// TIA Portal V20 export
FUNCTION_BLOCK "CallEquipment"   // FB21, LAD
TITLE = CallEquipment
AUTHOR : ERsystem_FA2_DH. Kim
// This block contains the logic and futher calls (e.g. sequences, control modules, diagnostics etc.) of the equipment module.
// stored: IsIECCheckEnabled true, MemoryReserve 100, Namespace Unit1.Em6, SetENOAutomatically false
   VAR_INPUT
      ZoneOperationEnable { ExternalWritable := 'False'} : "LWONIK_typeSafetyZoneManualOperation";
   END_VAR
   VAR_IN_OUT
      unitStatus : "LAF_typeUnitStatus";   // Current unit status o be used in this EM
      unitAlarmDB : "LAF_typeAlarms";   // Summarized EM Alarms for the Unit
      emFeedback : "LUC_typeEmFeedback";   // Feedback of the EM to the Unit
   END_VAR
   VAR
      InstSequenceStackTable { S7_SetPoint := 'True'} : "Unit1.Em6.Sequence_1_StackTable";
      InstSequenceGaugeRnR { S7_SetPoint := 'True'} : "Unit1.Em6.Sequence_10_GaugeRnR";
      InstSequenceUtility { S7_SetPoint := 'True'} : "Unit1.Em6.Sequence_20_Utility";
      instStackTableHomeJob1 { S7_SetPoint := 'True'} : "LAF_SelectJob";
      instStackTableMotionAutoJob2 { S7_SetPoint := 'True'} : "LAF_SelectJob";
      instStackTableRollerMoveJob12 { S7_SetPoint := 'True'} : "LAF_SelectJob";
      instStackTableRollerMoveJob13 { S7_SetPoint := 'True'} : "LAF_SelectJob";
      instStackTableAnodeMendrelJob22 { S7_SetPoint := 'True'} : "LAF_SelectJob";
      instStackTableCathodeMendrelJob23 { S7_SetPoint := 'True'} : "LAF_SelectJob";
      instStackTableVisionJob30 { S7_SetPoint := 'True'} : "LAF_SelectJob";
      instStackTableDownJob31 { S7_SetPoint := 'True'} : "LAF_SelectJob";
      instStackTableUnloadJob4 { S7_SetPoint := 'True'} : "LAF_SelectJob";
      instGaugeRnRReadyJob1 { S7_SetPoint := 'True'} : "LAF_SelectJob";
      instGaugeRnRVaccumJob2 { S7_SetPoint := 'True'} : "LAF_SelectJob";
      instGaugeRnRVisionJob3 { S7_SetPoint := 'True'} : "LAF_SelectJob";
      instGaugeRnRBlowJob4 { S7_SetPoint := 'True'} : "LAF_SelectJob";
      instUtilityFinalRollerHomeJob1 { S7_SetPoint := 'True'} : "LAF_SelectJob";
      instUtilityStackTableOutHomeJob2 { S7_SetPoint := 'True'} : "LAF_SelectJob";
      instUtilityAllMendrelOpenJob3 { S7_SetPoint := 'True'} : "LAF_SelectJob";
      instUtilityAllMendrelCloseJob4 { S7_SetPoint := 'True'} : "LAF_SelectJob";
      instCmStackTableElectrodeDetectSensor { S7_SetPoint := 'True'} : "LBC_DigitalSignalCn";
      instCmMasterVirtualAxisX : "LBC_Axis64Pos_TecPlcCn";
      instCmFinalRollerFrontAxisX : "LBC_Axis64Pos_TecPlcCn";
      instCmFinalRollerRearAxisX { S7_SetPoint := 'True'} : "LBC_Axis64Pos_TecPlcCn";
      instCmMendrelAnodeFrontAxisY { S7_SetPoint := 'True'} : "LBC_Axis64Pos_TecPlcCn";
      instCmMendrelAnodeFrontAxisZ { S7_SetPoint := 'True'} : "LBC_Axis64Pos_TecPlcCn";
      instCmMendrelAnodeRearAxisY { S7_SetPoint := 'True'} : "LBC_Axis64Pos_TecPlcCn";
      instCmMendrelAnodeRearAxisZ { S7_SetPoint := 'True'} : "LBC_Axis64Pos_TecPlcCn";
      instCmMendrelCathodeFrontAxisY { S7_SetPoint := 'True'} : "LBC_Axis64Pos_TecPlcCn";
      instCmMendrelCathodeFrontAxisZ { S7_SetPoint := 'True'} : "LBC_Axis64Pos_TecPlcCn";
      instCmMendrelCathodeRearAxisY { S7_SetPoint := 'True'} : "LBC_Axis64Pos_TecPlcCn";
      instCmMendrelCathodeRearAxisZ { S7_SetPoint := 'True'} : "LBC_Axis64Pos_TecPlcCn";
      instCmStackTableAxisZ { ExternalAccessible := 'False'; ExternalVisible := 'False'; ExternalWritable := 'False'; S7_SetPoint := 'True'} : "LBC_Axis64Pos_TecPlcCn";
      instCmStackTableOutFrontAxisZ { ExternalAccessible := 'False'; ExternalVisible := 'False'; ExternalWritable := 'False'; S7_SetPoint := 'True'} : "LBC_Axis64Pos_TecPlcCn";
      instCmStackTableOutRearAxisZ { ExternalAccessible := 'False'; ExternalVisible := 'False'; ExternalWritable := 'False'; S7_SetPoint := 'True'} : "LBC_Axis64Pos_TecPlcCn";
      instInterlockFinalRollerFrontAxisX : "LER_Axis64Pos_InterlockSummary";
      instInterlockFinalRollerRearAxisX : "LER_Axis64Pos_InterlockSummary";
      instInterlockMendrelAnodeFrontAxisY : "LER_Axis64Pos_InterlockSummary";
      instInterlockMendrelAnodeFrontAxisZ : "LER_Axis64Pos_InterlockSummary";
      instInterlockMendrelAnodeRearAxisY : "LER_Axis64Pos_InterlockSummary";
      instInterlockMendrelAnodeRearAxisZ : "LER_Axis64Pos_InterlockSummary";
      instInterlockMendrelCathodeFrontAxisY : "LER_Axis64Pos_InterlockSummary";
      instInterlockMendrelCathodeFrontAxisZ : "LER_Axis64Pos_InterlockSummary";
      instInterlockMendrelCathodeRearAxisY : "LER_Axis64Pos_InterlockSummary";
      instInterlockMendrelCathodeRearAxisZ : "LER_Axis64Pos_InterlockSummary";
      instInterlockStackTableAxisZ : "LER_Axis64Pos_InterlockSummary";
      instInterlockStackTableOutFrontAxisZ : "LER_Axis64Pos_InterlockSummary";
      instInterlockStackTableOutRearAxisZ : "LER_Axis64Pos_InterlockSummary";
      instFinalRollerFrontAxisXMCGearIn { S7_SetPoint := 'True'} : MC_GEARIN;
      instFinalRollerRearAxisXMCGearIn { S7_SetPoint := 'True'} : MC_GEARIN;
      instStackTableOutFrontAxisZMCGearIn { S7_SetPoint := 'True'} : MC_GEARIN;
      instStackTableOutRearAxisZMCGearIn { S7_SetPoint := 'True'} : MC_GEARIN;
      instFinalRollerFrontAxisXMCWirteParameter { S7_SetPoint := 'True'} : MC_WRITEPARAMETER;
      instFinalRollerRearAxisXMCWirteParameter { S7_SetPoint := 'True'} : MC_WRITEPARAMETER;
      instStackTableOutFrontAxisZMCWirteParameter { S7_SetPoint := 'True'} : MC_WRITEPARAMETER;
      instStackTableOutRearAxisZMCWirteParameter { S7_SetPoint := 'True'} : MC_WRITEPARAMETER;
      instCmMendrelCathodeFrontClamp { ExternalAccessible := 'False'; ExternalVisible := 'False'; ExternalWritable := 'False'; S7_SetPoint := 'True'} : "LBC_TwoWayActuatorCn";
      instCmMendrelAnodeFrontClamp { ExternalAccessible := 'False'; ExternalVisible := 'False'; ExternalWritable := 'False'; S7_SetPoint := 'True'} : "LBC_TwoWayActuatorCn";
      instCmMendrelCathodeRearClamp { ExternalAccessible := 'False'; ExternalVisible := 'False'; ExternalWritable := 'False'; S7_SetPoint := 'True'} : "LBC_TwoWayActuatorCn";
      instCmMendrelAnodeRearClamp { ExternalAccessible := 'False'; ExternalVisible := 'False'; ExternalWritable := 'False'; S7_SetPoint := 'True'} : "LBC_TwoWayActuatorCn";
      instcmStackTableVaccum { ExternalAccessible := 'False'; ExternalVisible := 'False'; ExternalWritable := 'False'; S7_SetPoint := 'True'} : "LBC_TwoWayActuatorCn";
      instcmStackTableGapPadUpDown { ExternalAccessible := 'False'; ExternalVisible := 'False'; ExternalWritable := 'False'; S7_SetPoint := 'True'} : "LBC_TwoWayActuatorCn";
      instCmStackTableVisionControllerInterface : "LER_Vision_XGX2000";
      instGapVisionConversion : "LER_StackTableVisionConversion";
      instManageAlarms { ExternalWritable := 'False'} : "LAF_ManageAlarms";
      instEventsPFE : "Unit1.Em6.EventsPFE";
      instLER_BrakeTestMendrelAnodeFrontAxisZ : "LER_BrakeTest";
      instLER_BrakeTestMendrelAnodeRearAxisZ { S7_SetPoint := 'True'} : "LER_BrakeTest";
      instLER_BrakeTestMendrelCathodeFrontAxisZ { S7_SetPoint := 'True'} : "LER_BrakeTest";
      instLER_BrakeTestMendrelCathodeRearAxisZ { S7_SetPoint := 'True'} : "LER_BrakeTest";
      instLER_BrakeTestStackTableAxisZ { S7_SetPoint := 'True'} : "LER_BrakeTest";
      instLER_BrakeTestStackTableOutFrontAxisZ { S7_SetPoint := 'True'} : "LER_BrakeTest";
      instLER_BrakeTestStackTableOutRearAxisZ { S7_SetPoint := 'True'} : "LER_BrakeTest";
      statUnitStatus { ExternalWritable := 'False'} : "LAF_typeUnitStatus";   // Unit Status used in this EM
      statSlmStatus : Struct
         running { ExternalWritable := 'False'} : Bool;
         powerOff { ExternalWritable := 'False'} : Bool;
      END_STRUCT;
      statAllBrakeTest { ExternalWritable := 'False'} : "LER_typeBrakeTestUnitCommands";
      statTonTime { ExternalAccessible := 'False'; ExternalVisible := 'False'; ExternalWritable := 'False'} : Array[0..1999] of TON_TIME;
      statTofTime { ExternalAccessible := 'False'; ExternalVisible := 'False'; ExternalWritable := 'False'} : Array[0..99] of TOF_TIME;
      statLReal { ExternalAccessible := 'False'; ExternalVisible := 'False'; ExternalWritable := 'False'} : Array[0..99] of LReal;
      statPulse { ExternalAccessible := 'False'; ExternalVisible := 'False'; ExternalWritable := 'False'} : Struct
         miscellaneous : Array[0..99] of Bool;
         workingDone : Array[0..99] of Bool;
         axisEnable : Array[0..99] of Bool;
         brakeTest : Array[0..99] of Bool;
      END_STRUCT;
      statEnableManualCmds : Bool;
      scan_on : Bool;
      "*** Interlock Axis ***" { ExternalAccessible := 'False'; ExternalVisible := 'False'; ExternalWritable := 'False'} : Bool;
      instFinalRollerFrontAxisX_CW { S7_SetPoint := 'True'} : "Jog.LER_Axis";
      instFinalRollerFrontAxisX_CCW { S7_SetPoint := 'True'} : "Jog.LER_Axis";
      instFinalRollerFrontAxisX_Home { S7_SetPoint := 'True'} : "Homing.LER_Axis";
      instFinalRollerFrontAxisX_Position { S7_SetPoint := 'True'} : Array[0..6] of "Position.LER_Axis";
      instFinalRollerRearAxisX_CW { S7_SetPoint := 'True'} : "Jog.LER_Axis";
      instFinalRollerRearAxisX_CCW { S7_SetPoint := 'True'} : "Jog.LER_Axis";
      instFinalRollerRearAxisX_Home { S7_SetPoint := 'True'} : "Homing.LER_Axis";
      instFinalRollerRearAxisX_Position { S7_SetPoint := 'True'} : Array[0..6] of "Position.LER_Axis";
      instMendrelAnodeFrontAxisY_CW { S7_SetPoint := 'True'} : "Jog.LER_Axis";
      instMendrelAnodeFrontAxisY_CCW { S7_SetPoint := 'True'} : "Jog.LER_Axis";
      instMendrelAnodeFrontAxisY_Home { S7_SetPoint := 'True'} : "Homing.LER_Axis";
      instMendrelAnodeFrontAxisY_Position { S7_SetPoint := 'True'} : Array[0..15] of "Position.LER_Axis";
      instMendrelAnodeFrontAxisZ_CW { S7_SetPoint := 'True'} : "Jog.LER_Axis";
      instMendrelAnodeFrontAxisZ_CCW { S7_SetPoint := 'True'} : "Jog.LER_Axis";
      instMendrelAnodeFrontAxisZ_Home { S7_SetPoint := 'True'} : "Homing.LER_Axis";
      instMendrelAnodeFrontAxisZ_Position { S7_SetPoint := 'True'} : Array[0..6] of "Position.LER_Axis";
      instMendrelAnodeRearAxisY_CW { S7_SetPoint := 'True'} : "Jog.LER_Axis";
      instMendrelAnodeRearAxisY_CCW { S7_SetPoint := 'True'} : "Jog.LER_Axis";
      instMendrelAnodeRearAxisY_Home { S7_SetPoint := 'True'} : "Homing.LER_Axis";
      instMendrelAnodeRearAxisY_Position { S7_SetPoint := 'True'} : Array[0..6] of "Position.LER_Axis";
      instMendrelAnodeRearAxisZ_CW { S7_SetPoint := 'True'} : "Jog.LER_Axis";
      instMendrelAnodeRearAxisZ_CCW { S7_SetPoint := 'True'} : "Jog.LER_Axis";
      instMendrelAnodeRearAxisZ_Home { S7_SetPoint := 'True'} : "Homing.LER_Axis";
      instMendrelAnodeRearAxisZ_Position { S7_SetPoint := 'True'} : Array[0..6] of "Position.LER_Axis";
      instMendrelCathodeFrontAxisY_CW { S7_SetPoint := 'True'} : "Jog.LER_Axis";
      instMendrelCathodeFrontAxisY_CCW { S7_SetPoint := 'True'} : "Jog.LER_Axis";
      instMendrelCathodeFrontAxisY_Home { S7_SetPoint := 'True'} : "Homing.LER_Axis";
      instMendrelCathodeFrontAxisY_Position { S7_SetPoint := 'True'} : Array[0..6] of "Position.LER_Axis";
      instMendrelCathodeFrontAxisZ_CW { S7_SetPoint := 'True'} : "Jog.LER_Axis";
      instMendrelCathodeFrontAxisZ_CCW { S7_SetPoint := 'True'} : "Jog.LER_Axis";
      instMendrelCathodeFrontAxisZ_Home { S7_SetPoint := 'True'} : "Homing.LER_Axis";
      instMendrelCathodeFrontAxisZ_Position { S7_SetPoint := 'True'} : Array[0..6] of "Position.LER_Axis";
      instMendrelCathodeRearAxisY_CW { S7_SetPoint := 'True'} : "Jog.LER_Axis";
      instMendrelCathodeRearAxisY_CCW { S7_SetPoint := 'True'} : "Jog.LER_Axis";
      instMendrelCathodeRearAxisY_Home { S7_SetPoint := 'True'} : "Homing.LER_Axis";
      instMendrelCathodeRearAxisY_Position { S7_SetPoint := 'True'} : Array[0..6] of "Position.LER_Axis";
      instMendrelCathodeRearAxisZ_CW { S7_SetPoint := 'True'} : "Jog.LER_Axis";
      instMendrelCathodeRearAxisZ_CCW { S7_SetPoint := 'True'} : "Jog.LER_Axis";
      instMendrelCathodeRearAxisZ_Home { S7_SetPoint := 'True'} : "Homing.LER_Axis";
      instMendrelCathodeRearAxisZ_Position { S7_SetPoint := 'True'} : Array[0..6] of "Position.LER_Axis";
      instStackTableAxisZ_CW { S7_SetPoint := 'True'} : "Jog.LER_Axis";
      instStackTableAxisZ_CCW { S7_SetPoint := 'True'} : "Jog.LER_Axis";
      instStackTableAxisZ_Home { S7_SetPoint := 'True'} : "Homing.LER_Axis";
      instStackTableAxisZ_Position { S7_SetPoint := 'True'} : Array[0..6] of "Position.LER_Axis";
      instStackTableOutFrontAxisZ_CW { S7_SetPoint := 'True'} : "Jog.LER_Axis";
      instStackTableOutFrontAxisZ_CCW { S7_SetPoint := 'True'} : "Jog.LER_Axis";
      instStackTableOutFrontAxisZ_Home { S7_SetPoint := 'True'} : "Homing.LER_Axis";
      instStackTableOutFrontAxisZ_Position { S7_SetPoint := 'True'} : Array[0..6] of "Position.LER_Axis";
      instStackTableOutRearAxisZ_CW { S7_SetPoint := 'True'} : "Jog.LER_Axis";
      instStackTableOutRearAxisZ_CCW { S7_SetPoint := 'True'} : "Jog.LER_Axis";
      instStackTableOutRearAxisZ_Home { S7_SetPoint := 'True'} : "Homing.LER_Axis";
      instStackTableOutRearAxisZ_Position { S7_SetPoint := 'True'} : Array[0..6] of "Position.LER_Axis";
      "*** Interlock Actuator ******" { ExternalAccessible := 'False'; ExternalVisible := 'False'; ExternalWritable := 'False'} : Bool;
      instCmMendrelCathodeFrontClampInterlock : Array[0..1] of "Cylinder.LER_Actuator";
      instCmMendrelAnodeFrontClampInterlock { S7_SetPoint := 'True'} : Array[0..1] of "Cylinder.LER_Actuator";
      instCmMendrelCathodeRearClampInterlock { S7_SetPoint := 'True'} : Array[0..1] of "Cylinder.LER_Actuator";
      instCmMendrelAnodeRearClampInterlock { S7_SetPoint := 'True'} : Array[0..1] of "Cylinder.LER_Actuator";
      instcmStackTableVaccumInterlock { S7_SetPoint := 'True'} : Array[0..1] of "Cylinder.LER_Actuator";
      instcmStackTableGapPadUpDownInterlock { S7_SetPoint := 'True'} : Array[0..1] of "Cylinder.LER_Actuator";
      AXIS21 : "LER_CM_Name";
      AXIS26 : "LER_CM_Name";
      AXIS31 : "LER_CM_Name";
      Cylinder33 : "LER_CM_Name";
      Vaccum20 : "LER_CM_Name";
      instFinalRollerGearInVel : MC_GEARINVELOCITY;
      instStackTableOutGearInVel : MC_GEARINVELOCITY;
      instFinalRollerGantryHoming : "LER_GantryHoming";
      instStackTableOutGantryHoming : "LER_GantryHoming";
      citi_Ptrig : Array[0..20] of Bool;
      citiTon : Array[0..20] of TON_TIME;
      citi : Time;
      citiTest : Array[0..20] of Bool;
   END_VAR
   VAR_TEMP
      tempIndex : Int;
      tempScInProduction : Bool;   // Mode Production and StateComplete
      tempScNoProduction : Bool;   // Mode Manual and StateComplete
   END_VAR
   VAR CONSTANT
      delayTime : Time := T#3s;
      TRUE : Bool := TRUE;
      FALSE : Bool := FALSE;
      NO_JOB : DInt;   // No job
      MIN_POSITION_NUMBER : SInt;
      INIT_POSITION_NUMBER : SInt := -1;
   END_VAR
   // // statPulse.brakeTest[0] : Unit Mode Production Rising Edge
   // // statPulse.brakeTest[1] : Unit Mode Production Rising Edge Old
   // // statPulse.brakeTest[10] : Mendrel Anode Front Z Axis Error Pulse
   // // statPulse.brakeTest[11] : Mendrel Anode Rear Z Axis Error Pulse
   // // statPulse.brakeTest[12] : Mendrel Cathode Front Z Axis Error Pulse
   // // statPulse.brakeTest[13] : Mendrel Cathode Rear Z Axis Error Pulse
   // // statPulse.brakeTest[14] : Stack Table Z Axis Error Pulse
   // // statPulse.brakeTest[15] : Stack Table Out Front Z Axis Error Pulse
   // // statPulse.brakeTest[16] : Stack Table Out Rear Z Axis Error Pulse
   VAR_TEMP   // added for the SCL form of the ladder/FBD networks
      _w1 : Bool;
      _w2 : Bool;
      _w3 : Bool;
      _w4 : Bool;
      _w5 : Bool;
      _w6 : Bool;
      _w7 : Bool;
      _w8 : Bool;
      _w9 : Bool;
      _w10 : Bool;
      _w11 : Bool;
   END_VAR
BEGIN

REGION Network 1: BLOCK INFO HEADER
   // (company) / (C) Copyright (year)
   // ---------------------------------------------------------------------------------
   // Title:                             (Title of this block)
   // Comment/Function: (that is implemented in the block)
   // Library/Family:           (that the source is dedicated to)
   // Author:                        (department / person in charge / contact)
   // Target System:          (test system with FW version)
   // Engineering:              TIA Portal (SW version)
   // Restrictions:               (OB types, etc.)
   // Requirements:           (hardware, technological package, etc.)
   // ---------------------------------------------------------------------------------
   // Change log table:
   // Version          | Date             | Signature      | Expert in charge  | Changes applied ------------------------|----------------------|-------------------------|--------------------------------|-----------------------
   // 001.000.000 | yyyy-mm-dd | 0x00000000 | (name of expert) | First released version
END_REGION

REGION Network 2: DESCRIPTION
   // This is a template block provided by the Automation Framework. It can be used to create an own project.
   // The Block Info Header is prepared to put in your own data.
   // Description of the block could be added here and the docu created by Code2Docu.
END_REGION

REGION Network 3: TRUE: Disable the monitoring of the Home position feedback. FALSE: Home position is reached after `monitoringReachingFeedback` time expires.
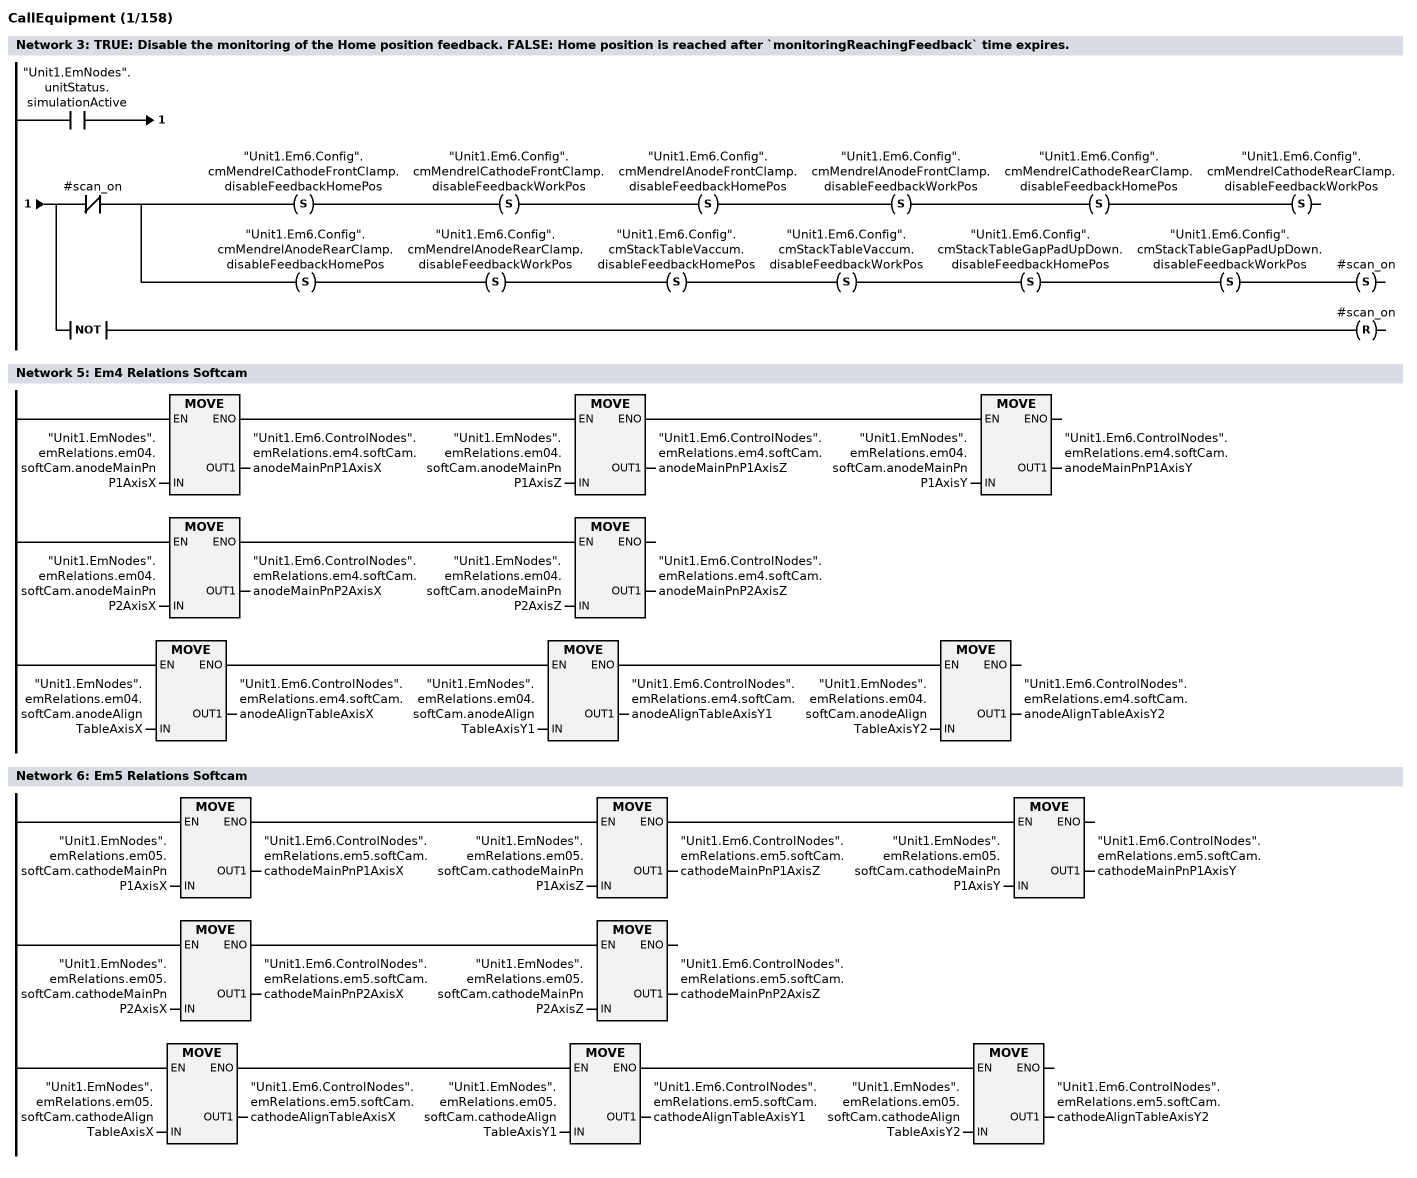
   RUNG wire#powerrail
      Contact( "Unit1.EmNodes".unitStatus.simulationActive )
      wire#w1
      I_Contact( #scan_on )
      wire#w2
      S_Coil( "Unit1.Em6.Config".cmMendrelCathodeFrontClamp.disableFeedbackHomePos )
      S_Coil( "Unit1.Em6.Config".cmMendrelCathodeFrontClamp.disableFeedbackWorkPos )
      S_Coil( "Unit1.Em6.Config".cmMendrelAnodeFrontClamp.disableFeedbackHomePos )
      S_Coil( "Unit1.Em6.Config".cmMendrelAnodeFrontClamp.disableFeedbackWorkPos )
      S_Coil( "Unit1.Em6.Config".cmMendrelCathodeRearClamp.disableFeedbackHomePos )
      S_Coil( "Unit1.Em6.Config".cmMendrelCathodeRearClamp.disableFeedbackWorkPos )
   END_RUNG
   RUNG wire#w2
      S_Coil( "Unit1.Em6.Config".cmMendrelAnodeRearClamp.disableFeedbackHomePos )
      S_Coil( "Unit1.Em6.Config".cmMendrelAnodeRearClamp.disableFeedbackWorkPos )
      S_Coil( "Unit1.Em6.Config".cmStackTableVaccum.disableFeedbackHomePos )
      S_Coil( "Unit1.Em6.Config".cmStackTableVaccum.disableFeedbackWorkPos )
      S_Coil( "Unit1.Em6.Config".cmStackTableGapPadUpDown.disableFeedbackHomePos )
      S_Coil( "Unit1.Em6.Config".cmStackTableGapPadUpDown.disableFeedbackWorkPos )
      S_Coil( #scan_on )
   END_RUNG
   RUNG wire#w1
      Not()
      R_Coil( #scan_on )
   END_RUNG
   // the same network as SCL:
   IF "Unit1.EmNodes".unitStatus.simulationActive AND NOT #scan_on THEN
       "Unit1.Em6.Config".cmMendrelCathodeFrontClamp.disableFeedbackHomePos := TRUE;
       "Unit1.Em6.Config".cmMendrelCathodeFrontClamp.disableFeedbackWorkPos := TRUE;
       "Unit1.Em6.Config".cmMendrelAnodeFrontClamp.disableFeedbackHomePos := TRUE;
       "Unit1.Em6.Config".cmMendrelAnodeFrontClamp.disableFeedbackWorkPos := TRUE;
       "Unit1.Em6.Config".cmMendrelCathodeRearClamp.disableFeedbackHomePos := TRUE;
       "Unit1.Em6.Config".cmMendrelCathodeRearClamp.disableFeedbackWorkPos := TRUE;
       "Unit1.Em6.Config".cmMendrelAnodeRearClamp.disableFeedbackHomePos := TRUE;
       "Unit1.Em6.Config".cmMendrelAnodeRearClamp.disableFeedbackWorkPos := TRUE;
       "Unit1.Em6.Config".cmStackTableVaccum.disableFeedbackHomePos := TRUE;
       "Unit1.Em6.Config".cmStackTableVaccum.disableFeedbackWorkPos := TRUE;
       "Unit1.Em6.Config".cmStackTableGapPadUpDown.disableFeedbackHomePos := TRUE;
       "Unit1.Em6.Config".cmStackTableGapPadUpDown.disableFeedbackWorkPos := TRUE;
       #scan_on := TRUE;
   END_IF;
   IF NOT "Unit1.EmNodes".unitStatus.simulationActive THEN #scan_on := FALSE; END_IF;
END_REGION

REGION Network 4: ******************** Unit Input ********************
END_REGION

REGION Network 5: Em4 Relations Softcam
   RUNG wire#powerrail
      Move(in := "Unit1.EmNodes".emRelations.em04.softCam.anodeMainPnP1AxisX, out1 => "Unit1.Em6.ControlNodes".emRelations.em4.softCam.anodeMainPnP1AxisX)
      Move(in := "Unit1.EmNodes".emRelations.em04.softCam.anodeMainPnP1AxisZ, out1 => "Unit1.Em6.ControlNodes".emRelations.em4.softCam.anodeMainPnP1AxisZ)
      Move(in := "Unit1.EmNodes".emRelations.em04.softCam.anodeMainPnP1AxisY, out1 => "Unit1.Em6.ControlNodes".emRelations.em4.softCam.anodeMainPnP1AxisY)
   END_RUNG
   RUNG wire#powerrail
      Move(in := "Unit1.EmNodes".emRelations.em04.softCam.anodeMainPnP2AxisX, out1 => "Unit1.Em6.ControlNodes".emRelations.em4.softCam.anodeMainPnP2AxisX)
      Move(in := "Unit1.EmNodes".emRelations.em04.softCam.anodeMainPnP2AxisZ, out1 => "Unit1.Em6.ControlNodes".emRelations.em4.softCam.anodeMainPnP2AxisZ)
   END_RUNG
   RUNG wire#powerrail
      Move(in := "Unit1.EmNodes".emRelations.em04.softCam.anodeAlignTableAxisX, out1 => "Unit1.Em6.ControlNodes".emRelations.em4.softCam.anodeAlignTableAxisX)
      Move(in := "Unit1.EmNodes".emRelations.em04.softCam.anodeAlignTableAxisY1, out1 => "Unit1.Em6.ControlNodes".emRelations.em4.softCam.anodeAlignTableAxisY1)
      Move(in := "Unit1.EmNodes".emRelations.em04.softCam.anodeAlignTableAxisY2, out1 => "Unit1.Em6.ControlNodes".emRelations.em4.softCam.anodeAlignTableAxisY2)
   END_RUNG
   // the same network as SCL:
   "Unit1.Em6.ControlNodes".emRelations.em4.softCam.anodeMainPnP1AxisX := "Unit1.EmNodes".emRelations.em04.softCam.anodeMainPnP1AxisX;
   "Unit1.Em6.ControlNodes".emRelations.em4.softCam.anodeMainPnP1AxisZ := "Unit1.EmNodes".emRelations.em04.softCam.anodeMainPnP1AxisZ;
   "Unit1.Em6.ControlNodes".emRelations.em4.softCam.anodeMainPnP1AxisY := "Unit1.EmNodes".emRelations.em04.softCam.anodeMainPnP1AxisY;
   "Unit1.Em6.ControlNodes".emRelations.em4.softCam.anodeMainPnP2AxisX := "Unit1.EmNodes".emRelations.em04.softCam.anodeMainPnP2AxisX;
   "Unit1.Em6.ControlNodes".emRelations.em4.softCam.anodeMainPnP2AxisZ := "Unit1.EmNodes".emRelations.em04.softCam.anodeMainPnP2AxisZ;
   "Unit1.Em6.ControlNodes".emRelations.em4.softCam.anodeAlignTableAxisX := "Unit1.EmNodes".emRelations.em04.softCam.anodeAlignTableAxisX;
   "Unit1.Em6.ControlNodes".emRelations.em4.softCam.anodeAlignTableAxisY1 := "Unit1.EmNodes".emRelations.em04.softCam.anodeAlignTableAxisY1;
   "Unit1.Em6.ControlNodes".emRelations.em4.softCam.anodeAlignTableAxisY2 := "Unit1.EmNodes".emRelations.em04.softCam.anodeAlignTableAxisY2;
END_REGION

REGION Network 6: Em5 Relations Softcam
   RUNG wire#powerrail
      Move(in := "Unit1.EmNodes".emRelations.em05.softCam.cathodeMainPnP1AxisX, out1 => "Unit1.Em6.ControlNodes".emRelations.em5.softCam.cathodeMainPnP1AxisX)
      Move(in := "Unit1.EmNodes".emRelations.em05.softCam.cathodeMainPnP1AxisZ, out1 => "Unit1.Em6.ControlNodes".emRelations.em5.softCam.cathodeMainPnP1AxisZ)
      Move(in := "Unit1.EmNodes".emRelations.em05.softCam.cathodeMainPnP1AxisY, out1 => "Unit1.Em6.ControlNodes".emRelations.em5.softCam.cathodeMainPnP1AxisY)
   END_RUNG
   RUNG wire#powerrail
      Move(in := "Unit1.EmNodes".emRelations.em05.softCam.cathodeMainPnP2AxisX, out1 => "Unit1.Em6.ControlNodes".emRelations.em5.softCam.cathodeMainPnP2AxisX)
      Move(in := "Unit1.EmNodes".emRelations.em05.softCam.cathodeMainPnP2AxisZ, out1 => "Unit1.Em6.ControlNodes".emRelations.em5.softCam.cathodeMainPnP2AxisZ)
   END_RUNG
   RUNG wire#powerrail
      Move(in := "Unit1.EmNodes".emRelations.em05.softCam.cathodeAlignTableAxisX, out1 => "Unit1.Em6.ControlNodes".emRelations.em5.softCam.cathodeAlignTableAxisX)
      Move(in := "Unit1.EmNodes".emRelations.em05.softCam.cathodeAlignTableAxisY1, out1 => "Unit1.Em6.ControlNodes".emRelations.em5.softCam.cathodeAlignTableAxisY1)
      Move(in := "Unit1.EmNodes".emRelations.em05.softCam.cathodeAlignTableAxisY2, out1 => "Unit1.Em6.ControlNodes".emRelations.em5.softCam.cathodeAlignTableAxisY2)
   END_RUNG
   // the same network as SCL:
   "Unit1.Em6.ControlNodes".emRelations.em5.softCam.cathodeMainPnP1AxisX := "Unit1.EmNodes".emRelations.em05.softCam.cathodeMainPnP1AxisX;
   "Unit1.Em6.ControlNodes".emRelations.em5.softCam.cathodeMainPnP1AxisZ := "Unit1.EmNodes".emRelations.em05.softCam.cathodeMainPnP1AxisZ;
   "Unit1.Em6.ControlNodes".emRelations.em5.softCam.cathodeMainPnP1AxisY := "Unit1.EmNodes".emRelations.em05.softCam.cathodeMainPnP1AxisY;
   "Unit1.Em6.ControlNodes".emRelations.em5.softCam.cathodeMainPnP2AxisX := "Unit1.EmNodes".emRelations.em05.softCam.cathodeMainPnP2AxisX;
   "Unit1.Em6.ControlNodes".emRelations.em5.softCam.cathodeMainPnP2AxisZ := "Unit1.EmNodes".emRelations.em05.softCam.cathodeMainPnP2AxisZ;
   "Unit1.Em6.ControlNodes".emRelations.em5.softCam.cathodeAlignTableAxisX := "Unit1.EmNodes".emRelations.em05.softCam.cathodeAlignTableAxisX;
   "Unit1.Em6.ControlNodes".emRelations.em5.softCam.cathodeAlignTableAxisY1 := "Unit1.EmNodes".emRelations.em05.softCam.cathodeAlignTableAxisY1;
   "Unit1.Em6.ControlNodes".emRelations.em5.softCam.cathodeAlignTableAxisY2 := "Unit1.EmNodes".emRelations.em05.softCam.cathodeAlignTableAxisY2;
END_REGION

REGION Network 7: Em7 Relations Softcam
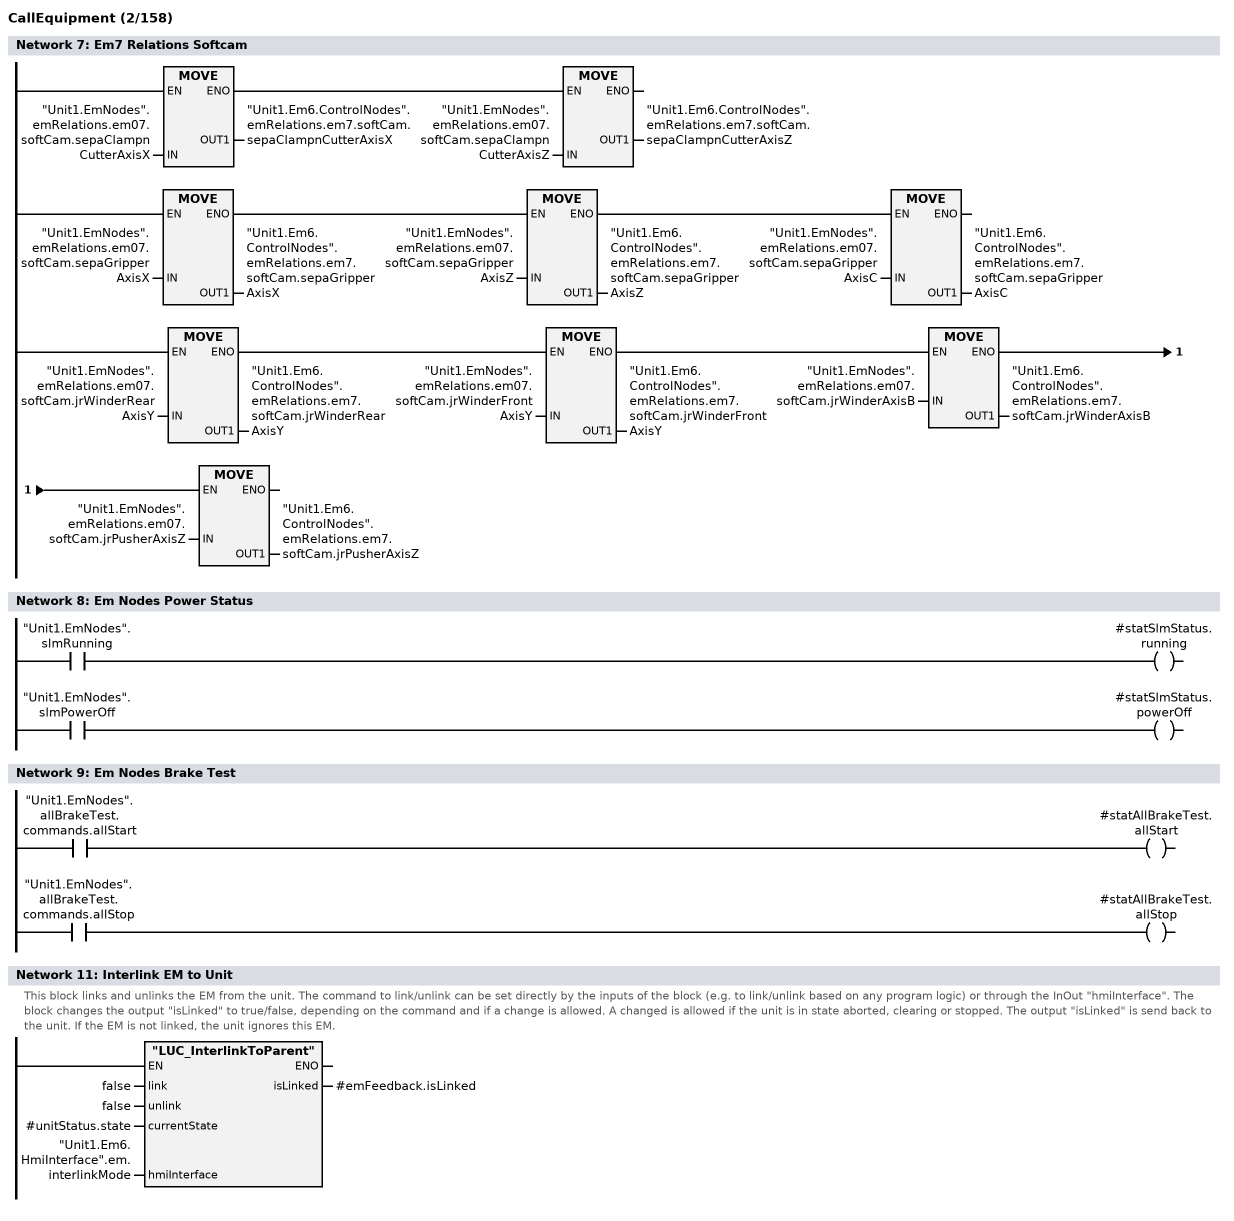
   RUNG wire#powerrail
      Move(in := "Unit1.EmNodes".emRelations.em07.softCam.sepaClampnCutterAxisX, out1 => "Unit1.Em6.ControlNodes".emRelations.em7.softCam.sepaClampnCutterAxisX)
      Move(in := "Unit1.EmNodes".emRelations.em07.softCam.sepaClampnCutterAxisZ, out1 => "Unit1.Em6.ControlNodes".emRelations.em7.softCam.sepaClampnCutterAxisZ)
   END_RUNG
   RUNG wire#powerrail
      Move(in := "Unit1.EmNodes".emRelations.em07.softCam.sepaGripperAxisX, out1 => "Unit1.Em6.ControlNodes".emRelations.em7.softCam.sepaGripperAxisX)
      Move(in := "Unit1.EmNodes".emRelations.em07.softCam.sepaGripperAxisZ, out1 => "Unit1.Em6.ControlNodes".emRelations.em7.softCam.sepaGripperAxisZ)
      Move(in := "Unit1.EmNodes".emRelations.em07.softCam.sepaGripperAxisC, out1 => "Unit1.Em6.ControlNodes".emRelations.em7.softCam.sepaGripperAxisC)
   END_RUNG
   RUNG wire#powerrail
      Move(in := "Unit1.EmNodes".emRelations.em07.softCam.jrWinderRearAxisY, out1 => "Unit1.Em6.ControlNodes".emRelations.em7.softCam.jrWinderRearAxisY)
      Move(in := "Unit1.EmNodes".emRelations.em07.softCam.jrWinderFrontAxisY, out1 => "Unit1.Em6.ControlNodes".emRelations.em7.softCam.jrWinderFrontAxisY)
      Move(in := "Unit1.EmNodes".emRelations.em07.softCam.jrWinderAxisB, out1 => "Unit1.Em6.ControlNodes".emRelations.em7.softCam.jrWinderAxisB)
      Move(in := "Unit1.EmNodes".emRelations.em07.softCam.jrPusherAxisZ, out1 => "Unit1.Em6.ControlNodes".emRelations.em7.softCam.jrPusherAxisZ)
   END_RUNG
   // the same network as SCL:
   "Unit1.Em6.ControlNodes".emRelations.em7.softCam.sepaClampnCutterAxisX := "Unit1.EmNodes".emRelations.em07.softCam.sepaClampnCutterAxisX;
   "Unit1.Em6.ControlNodes".emRelations.em7.softCam.sepaClampnCutterAxisZ := "Unit1.EmNodes".emRelations.em07.softCam.sepaClampnCutterAxisZ;
   "Unit1.Em6.ControlNodes".emRelations.em7.softCam.sepaGripperAxisX := "Unit1.EmNodes".emRelations.em07.softCam.sepaGripperAxisX;
   "Unit1.Em6.ControlNodes".emRelations.em7.softCam.sepaGripperAxisZ := "Unit1.EmNodes".emRelations.em07.softCam.sepaGripperAxisZ;
   "Unit1.Em6.ControlNodes".emRelations.em7.softCam.sepaGripperAxisC := "Unit1.EmNodes".emRelations.em07.softCam.sepaGripperAxisC;
   "Unit1.Em6.ControlNodes".emRelations.em7.softCam.jrWinderRearAxisY := "Unit1.EmNodes".emRelations.em07.softCam.jrWinderRearAxisY;
   "Unit1.Em6.ControlNodes".emRelations.em7.softCam.jrWinderFrontAxisY := "Unit1.EmNodes".emRelations.em07.softCam.jrWinderFrontAxisY;
   "Unit1.Em6.ControlNodes".emRelations.em7.softCam.jrWinderAxisB := "Unit1.EmNodes".emRelations.em07.softCam.jrWinderAxisB;
   "Unit1.Em6.ControlNodes".emRelations.em7.softCam.jrPusherAxisZ := "Unit1.EmNodes".emRelations.em07.softCam.jrPusherAxisZ;
END_REGION

REGION Network 8: Em Nodes Power Status
   RUNG wire#powerrail
      Contact( "Unit1.EmNodes".slmRunning )
      Coil( #statSlmStatus.running )
   END_RUNG
   RUNG wire#powerrail
      Contact( "Unit1.EmNodes".slmPowerOff )
      Coil( #statSlmStatus.powerOff )
   END_RUNG
   // the same network as SCL:
   #statSlmStatus.running := "Unit1.EmNodes".slmRunning;
   #statSlmStatus.powerOff := "Unit1.EmNodes".slmPowerOff;
END_REGION

REGION Network 9: Em Nodes Brake Test
   RUNG wire#powerrail
      Contact( "Unit1.EmNodes".allBrakeTest.commands.allStart )
      Coil( #statAllBrakeTest.allStart )
   END_RUNG
   RUNG wire#powerrail
      Contact( "Unit1.EmNodes".allBrakeTest.commands.allStop )
      Coil( #statAllBrakeTest.allStop )
   END_RUNG
   // the same network as SCL:
   #statAllBrakeTest.allStart := "Unit1.EmNodes".allBrakeTest.commands.allStart;
   #statAllBrakeTest.allStop := "Unit1.EmNodes".allBrakeTest.commands.allStop;
END_REGION

REGION Network 10: *************** Equipment Control **************************
END_REGION

REGION Network 11: Interlink EM to Unit
   // This block links and unlinks the EM from the unit. The command to link/unlink can be set directly by the inputs of the block (e.g. to link/unlink based on any program logic) or through the InOut "hmiInterface". The block changes the output "isLinked" to true/false, depending on the command and if a change is allowed. A changed is allowed if the unit is in state aborted, clearing or stopped. The output "isLinked" is send back to the unit. If the EM is not linked, the unit ignores this EM.
   RUNG wire#powerrail
      "LUC_InterlinkToParent"(link := false, unlink := false, currentState := #unitStatus.state, hmiInterface := "Unit1.Em6.HmiInterface".em.interlinkMode, isLinked => #emFeedback.isLinked)
   END_RUNG
   // the same network as SCL:
   "LUC_InterlinkToParent"(link := false,
                           unlink := false,
                           currentState := #unitStatus.state,
                           hmiInterface := "Unit1.Em6.HmiInterface".em.interlinkMode,
                           isLinked => #emFeedback.isLinked);
END_REGION

REGION Network 12: Control EM
   // When linked, unitStatus is fully applied to unitStatusUsed.
   // When not linked, only acknowledge and safetyReleased from the unitStatus are applied. A direct EM control by hmiInterface or localInterface is possible.
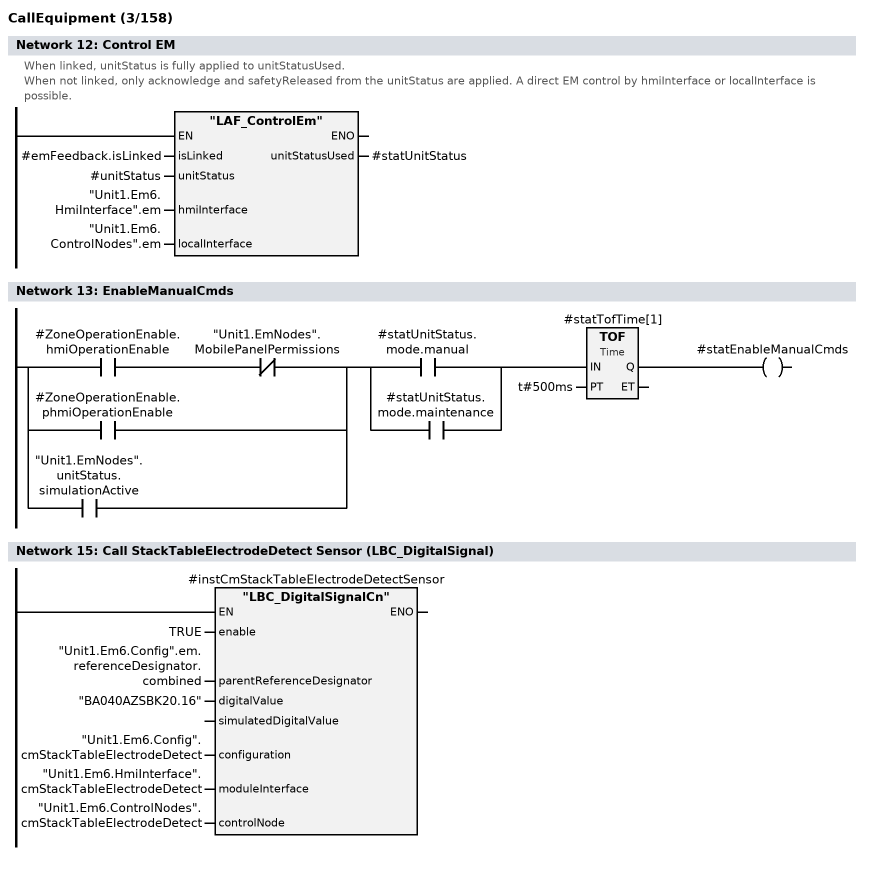
   RUNG wire#powerrail
      "LAF_ControlEm"(isLinked := #emFeedback.isLinked, unitStatus := #unitStatus, hmiInterface := "Unit1.Em6.HmiInterface".em, localInterface := "Unit1.Em6.ControlNodes".em, unitStatusUsed => #statUnitStatus)
   END_RUNG
   // the same network as SCL:
   "LAF_ControlEm"(isLinked := #emFeedback.isLinked,
                   unitStatus := #unitStatus,
                   hmiInterface := "Unit1.Em6.HmiInterface".em,
                   localInterface := "Unit1.Em6.ControlNodes".em,
                   unitStatusUsed => #statUnitStatus);
END_REGION

REGION Network 13: EnableManualCmds
   RUNG wire#powerrail
      Contact( #ZoneOperationEnable.hmiOperationEnable )
      I_Contact( "Unit1.EmNodes".MobilePanelPermissions )
      wire#w1
      Contact( #statUnitStatus.mode.manual )
      wire#w2
      { S7_Templates := "time_type := Time" } #statTofTime[1].TOF(pt := t#500ms, et =>)
      Coil( #statEnableManualCmds )
   END_RUNG
   RUNG wire#powerrail
      Contact( #ZoneOperationEnable.phmiOperationEnable )
   END_RUNG wire#w1
   RUNG wire#powerrail
      Contact( "Unit1.EmNodes".unitStatus.simulationActive )
   END_RUNG wire#w1
   RUNG wire#w1
      Contact( #statUnitStatus.mode.maintenance )
   END_RUNG wire#w2
   // the same network as SCL:
   #statTofTime[1].TOF(IN := ((#ZoneOperationEnable.hmiOperationEnable AND NOT "Unit1.EmNodes".MobilePanelPermissions) OR #ZoneOperationEnable.phmiOperationEnable OR "Unit1.EmNodes".unitStatus.simulationActive) AND (#statUnitStatus.mode.manual OR #statUnitStatus.mode.maintenance),
                       PT := t#500ms);
   #statEnableManualCmds := #statTofTime[1].Q;
END_REGION

REGION Network 14: *************** Control Modules (Sensors) ********************
   // Call control modules that are sensors before the em logic (jobs and sequence), so that the latest value is used in the logic.
END_REGION

REGION Network 15: Call StackTableElectrodeDetect Sensor (LBC_DigitalSignal)
   RUNG wire#powerrail
      #instCmStackTableElectrodeDetectSensor(enable := TRUE, parentReferenceDesignator := "Unit1.Em6.Config".em.referenceDesignator.combined, digitalValue := "BA040AZSBK20.16", simulatedDigitalValue :=, configuration := "Unit1.Em6.Config".cmStackTableElectrodeDetect, moduleInterface := "Unit1.Em6.HmiInterface".cmStackTableElectrodeDetect, controlNode := "Unit1.Em6.ControlNodes".cmStackTableElectrodeDetect)
   END_RUNG
   // the same network as SCL:
   #instCmStackTableElectrodeDetectSensor(enable := TRUE,   // "LBC_DigitalSignalCn"
                           parentReferenceDesignator := "Unit1.Em6.Config".em.referenceDesignator.combined,
                           digitalValue := "BA040AZSBK20.16",
                           configuration := "Unit1.Em6.Config".cmStackTableElectrodeDetect,
                           moduleInterface := "Unit1.Em6.HmiInterface".cmStackTableElectrodeDetect,
                           controlNode := "Unit1.Em6.ControlNodes".cmStackTableElectrodeDetect);
END_REGION

REGION Network 16: ******************** Equipment Logic ********************
END_REGION

REGION Network 17: Map Unit Status to Sequence Status [Step]
   // This block maps the unit status to the seuqnce status. Thus, it controls the sequence depending on the unit status. E.g. it sets the sequence to automatic when the unit state is in productions. This blocks work perfectly with the sequences provided in the AF. 
   // This typed block (MapUnitStatusToSequence) could be adjusted to specific application requirements or if other, user-defined sequences are used.
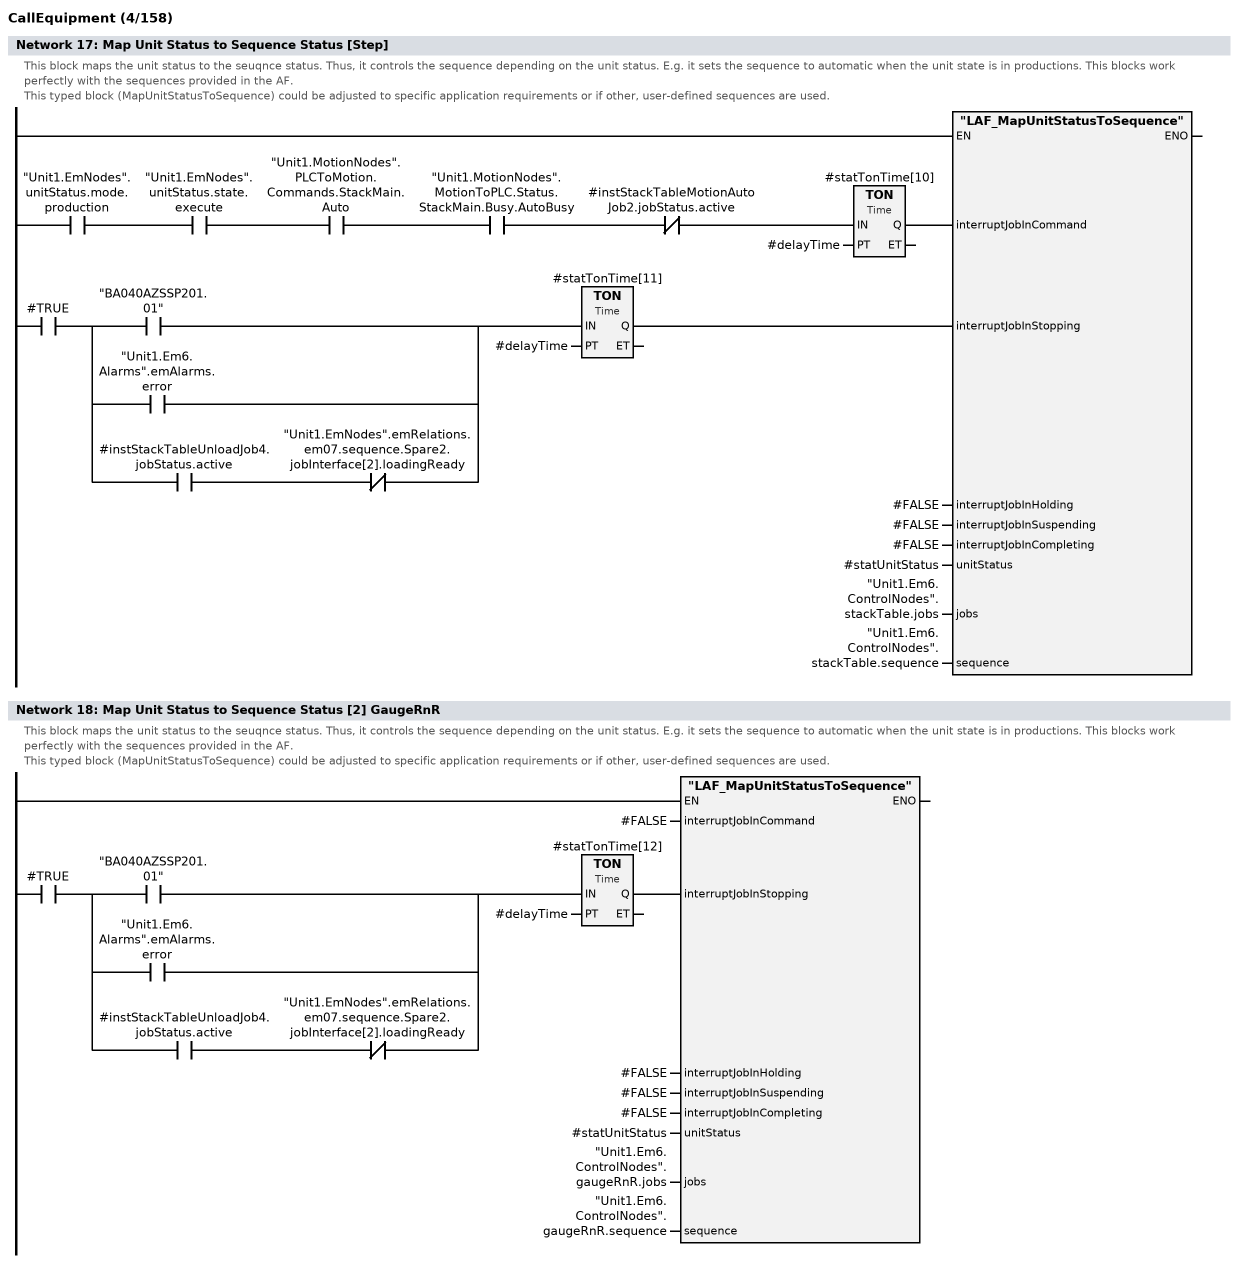
   RUNG wire#powerrail
      "LAF_MapUnitStatusToSequence"(interruptJobInCommand := wire#w1, interruptJobInStopping := wire#w4, interruptJobInHolding := #FALSE, interruptJobInSuspending := #FALSE, interruptJobInCompleting := #FALSE, unitStatus := #statUnitStatus, jobs := "Unit1.Em6.ControlNodes".stackTable.jobs, sequence := "Unit1.Em6.ControlNodes".stackTable.sequence)
   END_RUNG
   RUNG wire#powerrail
      Contact( "Unit1.EmNodes".unitStatus.mode.production )
      Contact( "Unit1.EmNodes".unitStatus.state.execute )
      Contact( "Unit1.MotionNodes".PLCToMotion.Commands.StackMain.Auto )
      Contact( "Unit1.MotionNodes".MotionToPLC.Status.StackMain.Busy.AutoBusy )
      I_Contact( #instStackTableMotionAutoJob2.jobStatus.active )
      { S7_Templates := "time_type := Time" } #statTonTime[10].TON(pt := #delayTime, et =>)
   END_RUNG wire#w1
   RUNG wire#powerrail
      Contact( #TRUE )
      wire#w2
      Contact( "BA040AZSSP201.01" )
      wire#w3
      { S7_Templates := "time_type := Time" } #statTonTime[11].TON(pt := #delayTime, et =>)
   END_RUNG wire#w4
   RUNG wire#w2
      Contact( "Unit1.Em6.Alarms".emAlarms.error )
   END_RUNG wire#w3
   RUNG wire#w2
      Contact( #instStackTableUnloadJob4.jobStatus.active )
      I_Contact( "Unit1.EmNodes".emRelations.em07.sequence.Spare2.jobInterface[2].loadingReady )
   END_RUNG wire#w3
   // the same network as SCL:
   #statTonTime[10].TON(IN := "Unit1.EmNodes".unitStatus.mode.production AND "Unit1.EmNodes".unitStatus.state.execute AND "Unit1.MotionNodes".PLCToMotion.Commands.StackMain.Auto AND "Unit1.MotionNodes".MotionToPLC.Status.StackMain.Busy.AutoBusy AND NOT #instStackTableMotionAutoJob2.jobStatus.active,
                        PT := #delayTime);
   #_w1 := #statTonTime[10].Q;
   #statTonTime[11].TON(IN := #TRUE AND ("BA040AZSSP201.01" OR "Unit1.Em6.Alarms".emAlarms.error OR (#instStackTableUnloadJob4.jobStatus.active AND NOT "Unit1.EmNodes".emRelations.em07.sequence.Spare2.jobInterface[2].loadingReady)),
                        PT := #delayTime);
   "LAF_MapUnitStatusToSequence"(interruptJobInCommand := #_w1,
                           interruptJobInStopping := #statTonTime[11].Q,
                           interruptJobInHolding := #FALSE,
                           interruptJobInSuspending := #FALSE,
                           interruptJobInCompleting := #FALSE,
                           unitStatus := #statUnitStatus,
                           jobs := "Unit1.Em6.ControlNodes".stackTable.jobs,
                           sequence := "Unit1.Em6.ControlNodes".stackTable.sequence);
END_REGION

REGION Network 18: Map Unit Status to Sequence Status [2] GaugeRnR
   // This block maps the unit status to the seuqnce status. Thus, it controls the sequence depending on the unit status. E.g. it sets the sequence to automatic when the unit state is in productions. This blocks work perfectly with the sequences provided in the AF. 
   // This typed block (MapUnitStatusToSequence) could be adjusted to specific application requirements or if other, user-defined sequences are used.
   RUNG wire#powerrail
      "LAF_MapUnitStatusToSequence"(interruptJobInStopping := wire#w3, interruptJobInCommand := #FALSE, interruptJobInHolding := #FALSE, interruptJobInSuspending := #FALSE, interruptJobInCompleting := #FALSE, unitStatus := #statUnitStatus, jobs := "Unit1.Em6.ControlNodes".gaugeRnR.jobs, sequence := "Unit1.Em6.ControlNodes".gaugeRnR.sequence)
   END_RUNG
   RUNG wire#powerrail
      Contact( #TRUE )
      wire#w1
      Contact( "BA040AZSSP201.01" )
      wire#w2
      { S7_Templates := "time_type := Time" } #statTonTime[12].TON(pt := #delayTime, et =>)
   END_RUNG wire#w3
   RUNG wire#w1
      Contact( "Unit1.Em6.Alarms".emAlarms.error )
   END_RUNG wire#w2
   RUNG wire#w1
      Contact( #instStackTableUnloadJob4.jobStatus.active )
      I_Contact( "Unit1.EmNodes".emRelations.em07.sequence.Spare2.jobInterface[2].loadingReady )
   END_RUNG wire#w2
   // the same network as SCL:
   #statTonTime[12].TON(IN := #TRUE AND ("BA040AZSSP201.01" OR "Unit1.Em6.Alarms".emAlarms.error OR (#instStackTableUnloadJob4.jobStatus.active AND NOT "Unit1.EmNodes".emRelations.em07.sequence.Spare2.jobInterface[2].loadingReady)),
                        PT := #delayTime);
   "LAF_MapUnitStatusToSequence"(interruptJobInCommand := #FALSE,
                           interruptJobInStopping := #statTonTime[12].Q,
                           interruptJobInHolding := #FALSE,
                           interruptJobInSuspending := #FALSE,
                           interruptJobInCompleting := #FALSE,
                           unitStatus := #statUnitStatus,
                           jobs := "Unit1.Em6.ControlNodes".gaugeRnR.jobs,
                           sequence := "Unit1.Em6.ControlNodes".gaugeRnR.sequence);
END_REGION

REGION Network 19: Map Unit Status to Sequence Status [3] Utility
   // This block maps the unit status to the seuqnce status. Thus, it controls the sequence depending on the unit status. E.g. it sets the sequence to automatic when the unit state is in productions. This blocks work perfectly with the sequences provided in the AF. 
   // This typed block (MapUnitStatusToSequence) could be adjusted to specific application requirements or if other, user-defined sequences are used.
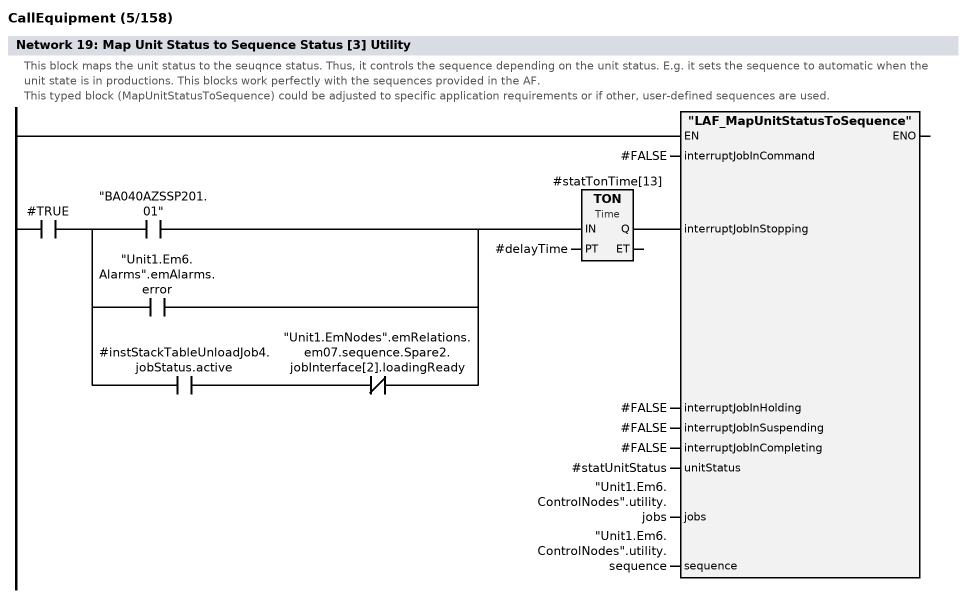
   RUNG wire#powerrail
      "LAF_MapUnitStatusToSequence"(interruptJobInStopping := wire#w3, interruptJobInCommand := #FALSE, interruptJobInHolding := #FALSE, interruptJobInSuspending := #FALSE, interruptJobInCompleting := #FALSE, unitStatus := #statUnitStatus, jobs := "Unit1.Em6.ControlNodes".utility.jobs, sequence := "Unit1.Em6.ControlNodes".utility.sequence)
   END_RUNG
   RUNG wire#powerrail
      Contact( #TRUE )
      wire#w1
      Contact( "BA040AZSSP201.01" )
      wire#w2
      { S7_Templates := "time_type := Time" } #statTonTime[13].TON(pt := #delayTime, et =>)
   END_RUNG wire#w3
   RUNG wire#w1
      Contact( "Unit1.Em6.Alarms".emAlarms.error )
   END_RUNG wire#w2
   RUNG wire#w1
      Contact( #instStackTableUnloadJob4.jobStatus.active )
      I_Contact( "Unit1.EmNodes".emRelations.em07.sequence.Spare2.jobInterface[2].loadingReady )
   END_RUNG wire#w2
   // the same network as SCL:
   #statTonTime[13].TON(IN := #TRUE AND ("BA040AZSSP201.01" OR "Unit1.Em6.Alarms".emAlarms.error OR (#instStackTableUnloadJob4.jobStatus.active AND NOT "Unit1.EmNodes".emRelations.em07.sequence.Spare2.jobInterface[2].loadingReady)),
                        PT := #delayTime);
   "LAF_MapUnitStatusToSequence"(interruptJobInCommand := #FALSE,
                           interruptJobInStopping := #statTonTime[13].Q,
                           interruptJobInHolding := #FALSE,
                           interruptJobInSuspending := #FALSE,
                           interruptJobInCompleting := #FALSE,
                           unitStatus := #statUnitStatus,
                           jobs := "Unit1.Em6.ControlNodes".utility.jobs,
                           sequence := "Unit1.Em6.ControlNodes".utility.sequence);
END_REGION

REGION Network 22: Select Job [GageRnR]
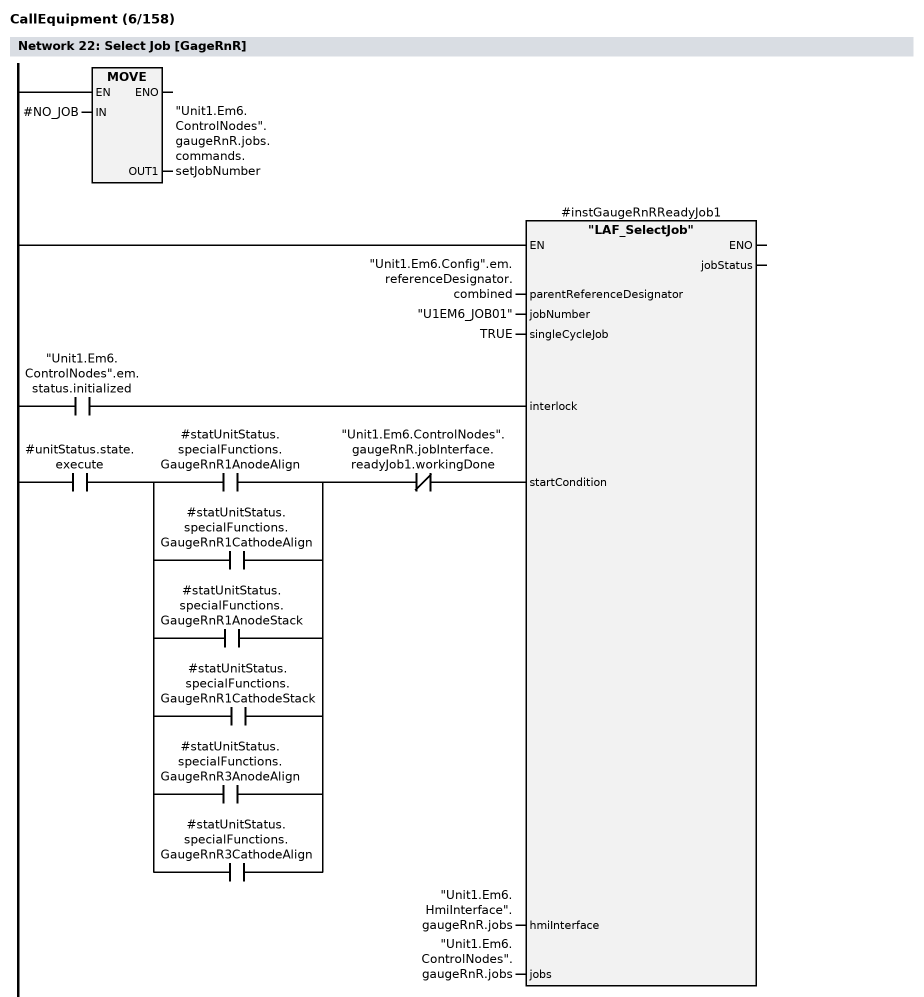
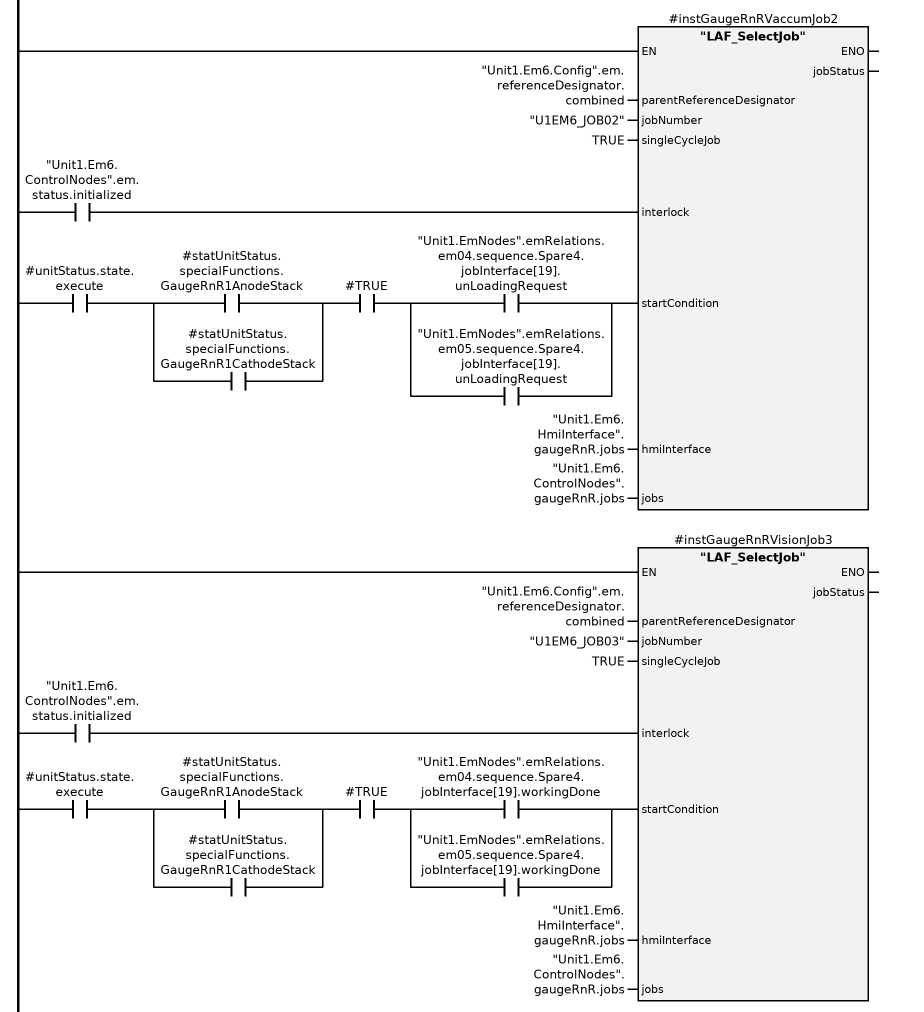
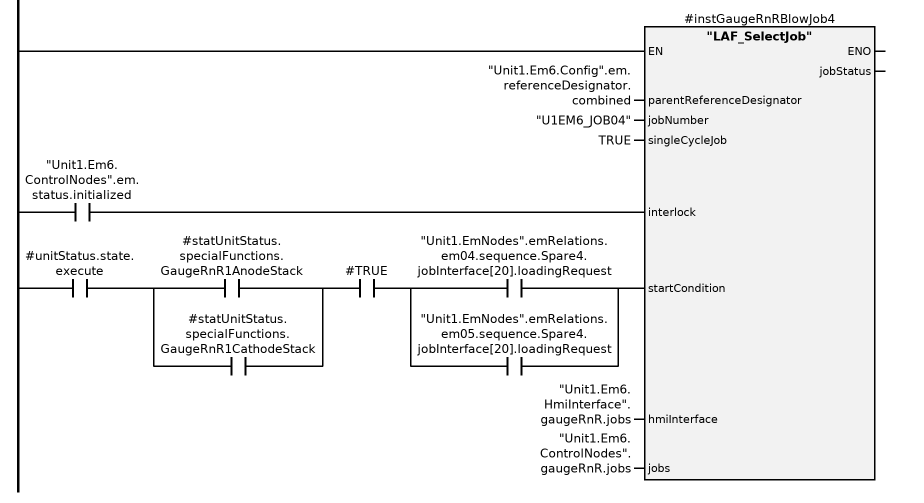
   RUNG wire#powerrail
      Move(in := #NO_JOB, out1 => "Unit1.Em6.ControlNodes".gaugeRnR.jobs.commands.setJobNumber)
   END_RUNG
   RUNG wire#powerrail
      #instGaugeRnRReadyJob1(interlock := wire#w1, startCondition := wire#w4, parentReferenceDesignator := "Unit1.Em6.Config".em.referenceDesignator.combined, jobNumber := "U1EM6_JOB01", singleCycleJob := TRUE, hmiInterface := "Unit1.Em6.HmiInterface".gaugeRnR.jobs, jobs := "Unit1.Em6.ControlNodes".gaugeRnR.jobs, jobStatus =>)
   END_RUNG
   RUNG wire#powerrail
      Contact( "Unit1.Em6.ControlNodes".em.status.initialized )
   END_RUNG wire#w1
   RUNG wire#powerrail
      Contact( #unitStatus.state.execute )
      wire#w2
      Contact( #statUnitStatus.specialFunctions.GaugeRnR1AnodeAlign )
      wire#w3
      I_Contact( "Unit1.Em6.ControlNodes".gaugeRnR.jobInterface.readyJob1.workingDone )
   END_RUNG wire#w4
   RUNG wire#w2
      Contact( #statUnitStatus.specialFunctions.GaugeRnR1CathodeAlign )
   END_RUNG wire#w3
   RUNG wire#w2
      Contact( #statUnitStatus.specialFunctions.GaugeRnR1AnodeStack )
   END_RUNG wire#w3
   RUNG wire#w2
      Contact( #statUnitStatus.specialFunctions.GaugeRnR1CathodeStack )
   END_RUNG wire#w3
   RUNG wire#w2
      Contact( #statUnitStatus.specialFunctions.GaugeRnR3AnodeAlign )
   END_RUNG wire#w3
   RUNG wire#w2
      Contact( #statUnitStatus.specialFunctions.GaugeRnR3CathodeAlign )
   END_RUNG wire#w3
   RUNG wire#powerrail
      #instGaugeRnRVaccumJob2(interlock := wire#w5, startCondition := wire#w9, parentReferenceDesignator := "Unit1.Em6.Config".em.referenceDesignator.combined, jobNumber := "U1EM6_JOB02", singleCycleJob := TRUE, hmiInterface := "Unit1.Em6.HmiInterface".gaugeRnR.jobs, jobs := "Unit1.Em6.ControlNodes".gaugeRnR.jobs, jobStatus =>)
   END_RUNG
   RUNG wire#powerrail
      Contact( "Unit1.Em6.ControlNodes".em.status.initialized )
   END_RUNG wire#w5
   RUNG wire#powerrail
      Contact( #unitStatus.state.execute )
      wire#w6
      Contact( #statUnitStatus.specialFunctions.GaugeRnR1AnodeStack )
      wire#w7
      Contact( #TRUE )
      wire#w8
      Contact( "Unit1.EmNodes".emRelations.em04.sequence.Spare4.jobInterface[19].unLoadingRequest )
   END_RUNG wire#w9
   RUNG wire#w6
      Contact( #statUnitStatus.specialFunctions.GaugeRnR1CathodeStack )
   END_RUNG wire#w7
   RUNG wire#w8
      Contact( "Unit1.EmNodes".emRelations.em05.sequence.Spare4.jobInterface[19].unLoadingRequest )
   END_RUNG wire#w9
   RUNG wire#powerrail
      #instGaugeRnRVisionJob3(interlock := wire#w10, startCondition := wire#w14, parentReferenceDesignator := "Unit1.Em6.Config".em.referenceDesignator.combined, jobNumber := "U1EM6_JOB03", singleCycleJob := TRUE, hmiInterface := "Unit1.Em6.HmiInterface".gaugeRnR.jobs, jobs := "Unit1.Em6.ControlNodes".gaugeRnR.jobs, jobStatus =>)
   END_RUNG
   RUNG wire#powerrail
      Contact( "Unit1.Em6.ControlNodes".em.status.initialized )
   END_RUNG wire#w10
   RUNG wire#powerrail
      Contact( #unitStatus.state.execute )
      wire#w11
      Contact( #statUnitStatus.specialFunctions.GaugeRnR1AnodeStack )
      wire#w12
      Contact( #TRUE )
      wire#w13
      Contact( "Unit1.EmNodes".emRelations.em04.sequence.Spare4.jobInterface[19].workingDone )
   END_RUNG wire#w14
   RUNG wire#w11
      Contact( #statUnitStatus.specialFunctions.GaugeRnR1CathodeStack )
   END_RUNG wire#w12
   RUNG wire#w13
      Contact( "Unit1.EmNodes".emRelations.em05.sequence.Spare4.jobInterface[19].workingDone )
   END_RUNG wire#w14
   RUNG wire#powerrail
      #instGaugeRnRBlowJob4(interlock := wire#w15, startCondition := wire#w19, parentReferenceDesignator := "Unit1.Em6.Config".em.referenceDesignator.combined, jobNumber := "U1EM6_JOB04", singleCycleJob := TRUE, hmiInterface := "Unit1.Em6.HmiInterface".gaugeRnR.jobs, jobs := "Unit1.Em6.ControlNodes".gaugeRnR.jobs, jobStatus =>)
   END_RUNG
   RUNG wire#powerrail
      Contact( "Unit1.Em6.ControlNodes".em.status.initialized )
   END_RUNG wire#w15
   RUNG wire#powerrail
      Contact( #unitStatus.state.execute )
      wire#w16
      Contact( #statUnitStatus.specialFunctions.GaugeRnR1AnodeStack )
      wire#w17
      Contact( #TRUE )
      wire#w18
      Contact( "Unit1.EmNodes".emRelations.em04.sequence.Spare4.jobInterface[20].loadingRequest )
   END_RUNG wire#w19
   RUNG wire#w16
      Contact( #statUnitStatus.specialFunctions.GaugeRnR1CathodeStack )
   END_RUNG wire#w17
   RUNG wire#w18
      Contact( "Unit1.EmNodes".emRelations.em05.sequence.Spare4.jobInterface[20].loadingRequest )
   END_RUNG wire#w19
   // the same network as SCL:
   "Unit1.Em6.ControlNodes".gaugeRnR.jobs.commands.setJobNumber := #NO_JOB;
   #instGaugeRnRReadyJob1(parentReferenceDesignator := "Unit1.Em6.Config".em.referenceDesignator.combined,   // "LAF_SelectJob"
                          jobNumber := "U1EM6_JOB01",
                          singleCycleJob := TRUE,
                          interlock := "Unit1.Em6.ControlNodes".em.status.initialized,
                          startCondition := #unitStatus.state.execute AND (#statUnitStatus.specialFunctions.GaugeRnR1AnodeAlign OR #statUnitStatus.specialFunctions.GaugeRnR1CathodeAlign OR #statUnitStatus.specialFunctions.GaugeRnR1AnodeStack OR #statUnitStatus.specialFunctions.GaugeRnR1CathodeStack OR #statUnitStatus.specialFunctions.GaugeRnR3AnodeAlign OR #statUnitStatus.specialFunctions.GaugeRnR3CathodeAlign) AND NOT "Unit1.Em6.ControlNodes".gaugeRnR.jobInterface.readyJob1.workingDone,
                          hmiInterface := "Unit1.Em6.HmiInterface".gaugeRnR.jobs,
                          jobs := "Unit1.Em6.ControlNodes".gaugeRnR.jobs);
   #instGaugeRnRVaccumJob2(parentReferenceDesignator := "Unit1.Em6.Config".em.referenceDesignator.combined,   // "LAF_SelectJob"
                           jobNumber := "U1EM6_JOB02",
                           singleCycleJob := TRUE,
                           interlock := "Unit1.Em6.ControlNodes".em.status.initialized,
                           startCondition := #unitStatus.state.execute AND (#statUnitStatus.specialFunctions.GaugeRnR1AnodeStack OR #statUnitStatus.specialFunctions.GaugeRnR1CathodeStack) AND #TRUE AND ("Unit1.EmNodes".emRelations.em04.sequence.Spare4.jobInterface[19].unLoadingRequest OR "Unit1.EmNodes".emRelations.em05.sequence.Spare4.jobInterface[19].unLoadingRequest),
                           hmiInterface := "Unit1.Em6.HmiInterface".gaugeRnR.jobs,
                           jobs := "Unit1.Em6.ControlNodes".gaugeRnR.jobs);
   #instGaugeRnRVisionJob3(parentReferenceDesignator := "Unit1.Em6.Config".em.referenceDesignator.combined,   // "LAF_SelectJob"
                           jobNumber := "U1EM6_JOB03",
                           singleCycleJob := TRUE,
                           interlock := "Unit1.Em6.ControlNodes".em.status.initialized,
                           startCondition := #unitStatus.state.execute AND (#statUnitStatus.specialFunctions.GaugeRnR1AnodeStack OR #statUnitStatus.specialFunctions.GaugeRnR1CathodeStack) AND #TRUE AND ("Unit1.EmNodes".emRelations.em04.sequence.Spare4.jobInterface[19].workingDone OR "Unit1.EmNodes".emRelations.em05.sequence.Spare4.jobInterface[19].workingDone),
                           hmiInterface := "Unit1.Em6.HmiInterface".gaugeRnR.jobs,
                           jobs := "Unit1.Em6.ControlNodes".gaugeRnR.jobs);
   #instGaugeRnRBlowJob4(parentReferenceDesignator := "Unit1.Em6.Config".em.referenceDesignator.combined,   // "LAF_SelectJob"
                         jobNumber := "U1EM6_JOB04",
                         singleCycleJob := TRUE,
                         interlock := "Unit1.Em6.ControlNodes".em.status.initialized,
                         startCondition := #unitStatus.state.execute AND (#statUnitStatus.specialFunctions.GaugeRnR1AnodeStack OR #statUnitStatus.specialFunctions.GaugeRnR1CathodeStack) AND #TRUE AND ("Unit1.EmNodes".emRelations.em04.sequence.Spare4.jobInterface[20].loadingRequest OR "Unit1.EmNodes".emRelations.em05.sequence.Spare4.jobInterface[20].loadingRequest),
                         hmiInterface := "Unit1.Em6.HmiInterface".gaugeRnR.jobs,
                         jobs := "Unit1.Em6.ControlNodes".gaugeRnR.jobs);
END_REGION

REGION Network 23: Stack Table Select Job [01] Initialize
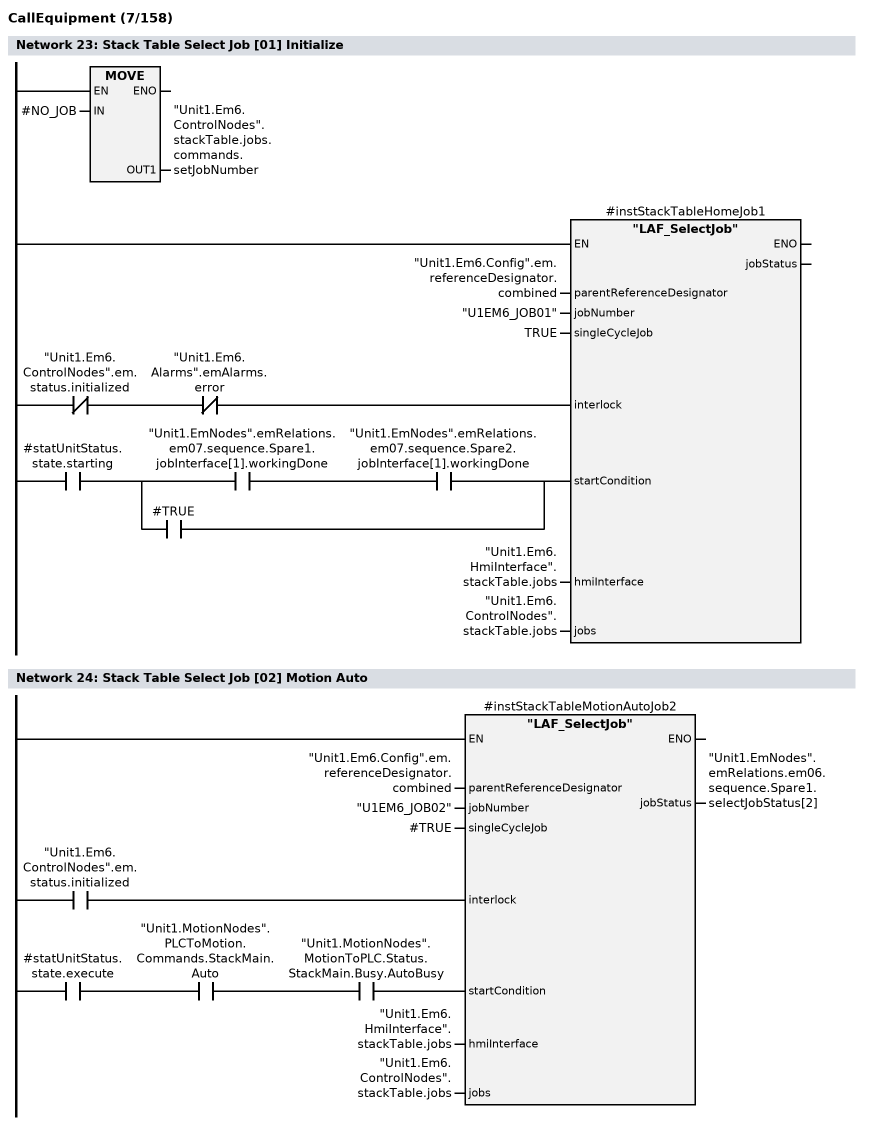
   RUNG wire#powerrail
      Move(in := #NO_JOB, out1 => "Unit1.Em6.ControlNodes".stackTable.jobs.commands.setJobNumber)
   END_RUNG
   RUNG wire#powerrail
      #instStackTableHomeJob1(interlock := wire#w1, startCondition := wire#w3, parentReferenceDesignator := "Unit1.Em6.Config".em.referenceDesignator.combined, jobNumber := "U1EM6_JOB01", singleCycleJob := TRUE, hmiInterface := "Unit1.Em6.HmiInterface".stackTable.jobs, jobs := "Unit1.Em6.ControlNodes".stackTable.jobs, jobStatus =>)
   END_RUNG
   RUNG wire#powerrail
      I_Contact( "Unit1.Em6.ControlNodes".em.status.initialized )
      I_Contact( "Unit1.Em6.Alarms".emAlarms.error )
   END_RUNG wire#w1
   RUNG wire#powerrail
      Contact( #statUnitStatus.state.starting )
      wire#w2
      Contact( "Unit1.EmNodes".emRelations.em07.sequence.Spare1.jobInterface[1].workingDone )
      Contact( "Unit1.EmNodes".emRelations.em07.sequence.Spare2.jobInterface[1].workingDone )
   END_RUNG wire#w3
   RUNG wire#w2
      Contact( #TRUE )
   END_RUNG wire#w3
   // the same network as SCL:
   "Unit1.Em6.ControlNodes".stackTable.jobs.commands.setJobNumber := #NO_JOB;
   #instStackTableHomeJob1(parentReferenceDesignator := "Unit1.Em6.Config".em.referenceDesignator.combined,   // "LAF_SelectJob"
                           jobNumber := "U1EM6_JOB01",
                           singleCycleJob := TRUE,
                           interlock := NOT "Unit1.Em6.ControlNodes".em.status.initialized AND NOT "Unit1.Em6.Alarms".emAlarms.error,
                           startCondition := #statUnitStatus.state.starting AND (("Unit1.EmNodes".emRelations.em07.sequence.Spare1.jobInterface[1].workingDone AND "Unit1.EmNodes".emRelations.em07.sequence.Spare2.jobInterface[1].workingDone) OR #TRUE),
                           hmiInterface := "Unit1.Em6.HmiInterface".stackTable.jobs,
                           jobs := "Unit1.Em6.ControlNodes".stackTable.jobs);
END_REGION

REGION Network 24: Stack Table Select Job [02] Motion Auto
   RUNG wire#powerrail
      #instStackTableMotionAutoJob2(interlock := wire#w1, startCondition := wire#w2, parentReferenceDesignator := "Unit1.Em6.Config".em.referenceDesignator.combined, jobNumber := "U1EM6_JOB02", singleCycleJob := #TRUE, hmiInterface := "Unit1.Em6.HmiInterface".stackTable.jobs, jobs := "Unit1.Em6.ControlNodes".stackTable.jobs, jobStatus => "Unit1.EmNodes".emRelations.em06.sequence.Spare1.selectJobStatus[2])
   END_RUNG
   RUNG wire#powerrail
      Contact( "Unit1.Em6.ControlNodes".em.status.initialized )
   END_RUNG wire#w1
   RUNG wire#powerrail
      Contact( #statUnitStatus.state.execute )
      Contact( "Unit1.MotionNodes".PLCToMotion.Commands.StackMain.Auto )
      Contact( "Unit1.MotionNodes".MotionToPLC.Status.StackMain.Busy.AutoBusy )
   END_RUNG wire#w2
   // the same network as SCL:
   #instStackTableMotionAutoJob2(parentReferenceDesignator := "Unit1.Em6.Config".em.referenceDesignator.combined,   // "LAF_SelectJob"
                           jobNumber := "U1EM6_JOB02",
                           singleCycleJob := #TRUE,
                           interlock := "Unit1.Em6.ControlNodes".em.status.initialized,
                           startCondition := #statUnitStatus.state.execute AND "Unit1.MotionNodes".PLCToMotion.Commands.StackMain.Auto AND "Unit1.MotionNodes".MotionToPLC.Status.StackMain.Busy.AutoBusy,
                           hmiInterface := "Unit1.Em6.HmiInterface".stackTable.jobs,
                           jobs := "Unit1.Em6.ControlNodes".stackTable.jobs,
                           jobStatus => "Unit1.EmNodes".emRelations.em06.sequence.Spare1.selectJobStatus[2]);
END_REGION

REGION Network 25: Stack Table Select Job [12] Final Roller Move Cathode → Anode
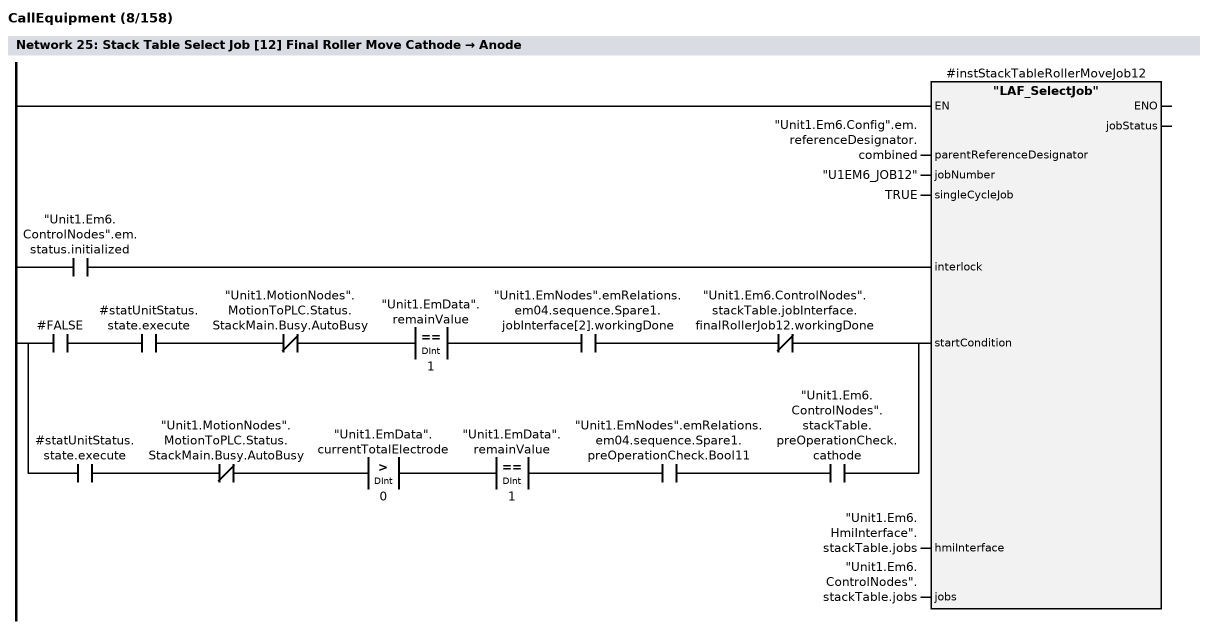
   RUNG wire#powerrail
      #instStackTableRollerMoveJob12(interlock := wire#w1, startCondition := wire#w2, parentReferenceDesignator := "Unit1.Em6.Config".em.referenceDesignator.combined, jobNumber := "U1EM6_JOB12", singleCycleJob := TRUE, hmiInterface := "Unit1.Em6.HmiInterface".stackTable.jobs, jobs := "Unit1.Em6.ControlNodes".stackTable.jobs, jobStatus =>)
   END_RUNG
   RUNG wire#powerrail
      Contact( "Unit1.Em6.ControlNodes".em.status.initialized )
   END_RUNG wire#w1
   RUNG wire#powerrail
      Contact( #FALSE )
      Contact( #statUnitStatus.state.execute )
      I_Contact( "Unit1.MotionNodes".MotionToPLC.Status.StackMain.Busy.AutoBusy )
      { S7_Templates := "SrcType := DInt" } EQ_Contact(in1 := "Unit1.EmData".remainValue, in2 := 1)
      Contact( "Unit1.EmNodes".emRelations.em04.sequence.Spare1.jobInterface[2].workingDone )
      I_Contact( "Unit1.Em6.ControlNodes".stackTable.jobInterface.finalRollerJob12.workingDone )
   END_RUNG wire#w2
   RUNG wire#powerrail
      Contact( #statUnitStatus.state.execute )
      I_Contact( "Unit1.MotionNodes".MotionToPLC.Status.StackMain.Busy.AutoBusy )
      { S7_Templates := "SrcType := DInt" } GT_Contact(in1 := "Unit1.EmData".currentTotalElectrode, in2 := 0)
      { S7_Templates := "SrcType := DInt" } EQ_Contact(in1 := "Unit1.EmData".remainValue, in2 := 1)
      Contact( "Unit1.EmNodes".emRelations.em04.sequence.Spare1.preOperationCheck.Bool11 )
      Contact( "Unit1.Em6.ControlNodes".stackTable.preOperationCheck.cathode )
   END_RUNG wire#w2
   // the same network as SCL:
   #instStackTableRollerMoveJob12(parentReferenceDesignator := "Unit1.Em6.Config".em.referenceDesignator.combined,   // "LAF_SelectJob"
                           jobNumber := "U1EM6_JOB12",
                           singleCycleJob := TRUE,
                           interlock := "Unit1.Em6.ControlNodes".em.status.initialized,
                           startCondition := (#FALSE AND #statUnitStatus.state.execute AND NOT "Unit1.MotionNodes".MotionToPLC.Status.StackMain.Busy.AutoBusy AND ("Unit1.EmData".remainValue = 1) AND "Unit1.EmNodes".emRelations.em04.sequence.Spare1.jobInterface[2].workingDone AND NOT "Unit1.Em6.ControlNodes".stackTable.jobInterface.finalRollerJob12.workingDone) OR (#statUnitStatus.state.execute AND NOT "Unit1.MotionNodes".MotionToPLC.Status.StackMain.Busy.AutoBusy AND ("Unit1.EmData".currentTotalElectrode > 0) AND ("Unit1.EmData".remainValue = 1) AND "Unit1.EmNodes".emRelations.em04.sequence.Spare1.preOperationCheck.Bool11 AND "Unit1.Em6.ControlNodes".stackTable.preOperationCheck.cathode),
                           hmiInterface := "Unit1.Em6.HmiInterface".stackTable.jobs,
                           jobs := "Unit1.Em6.ControlNodes".stackTable.jobs);
END_REGION

REGION Network 26: Stack Table Select Job [13] Final Roller Move Anode → Cathode
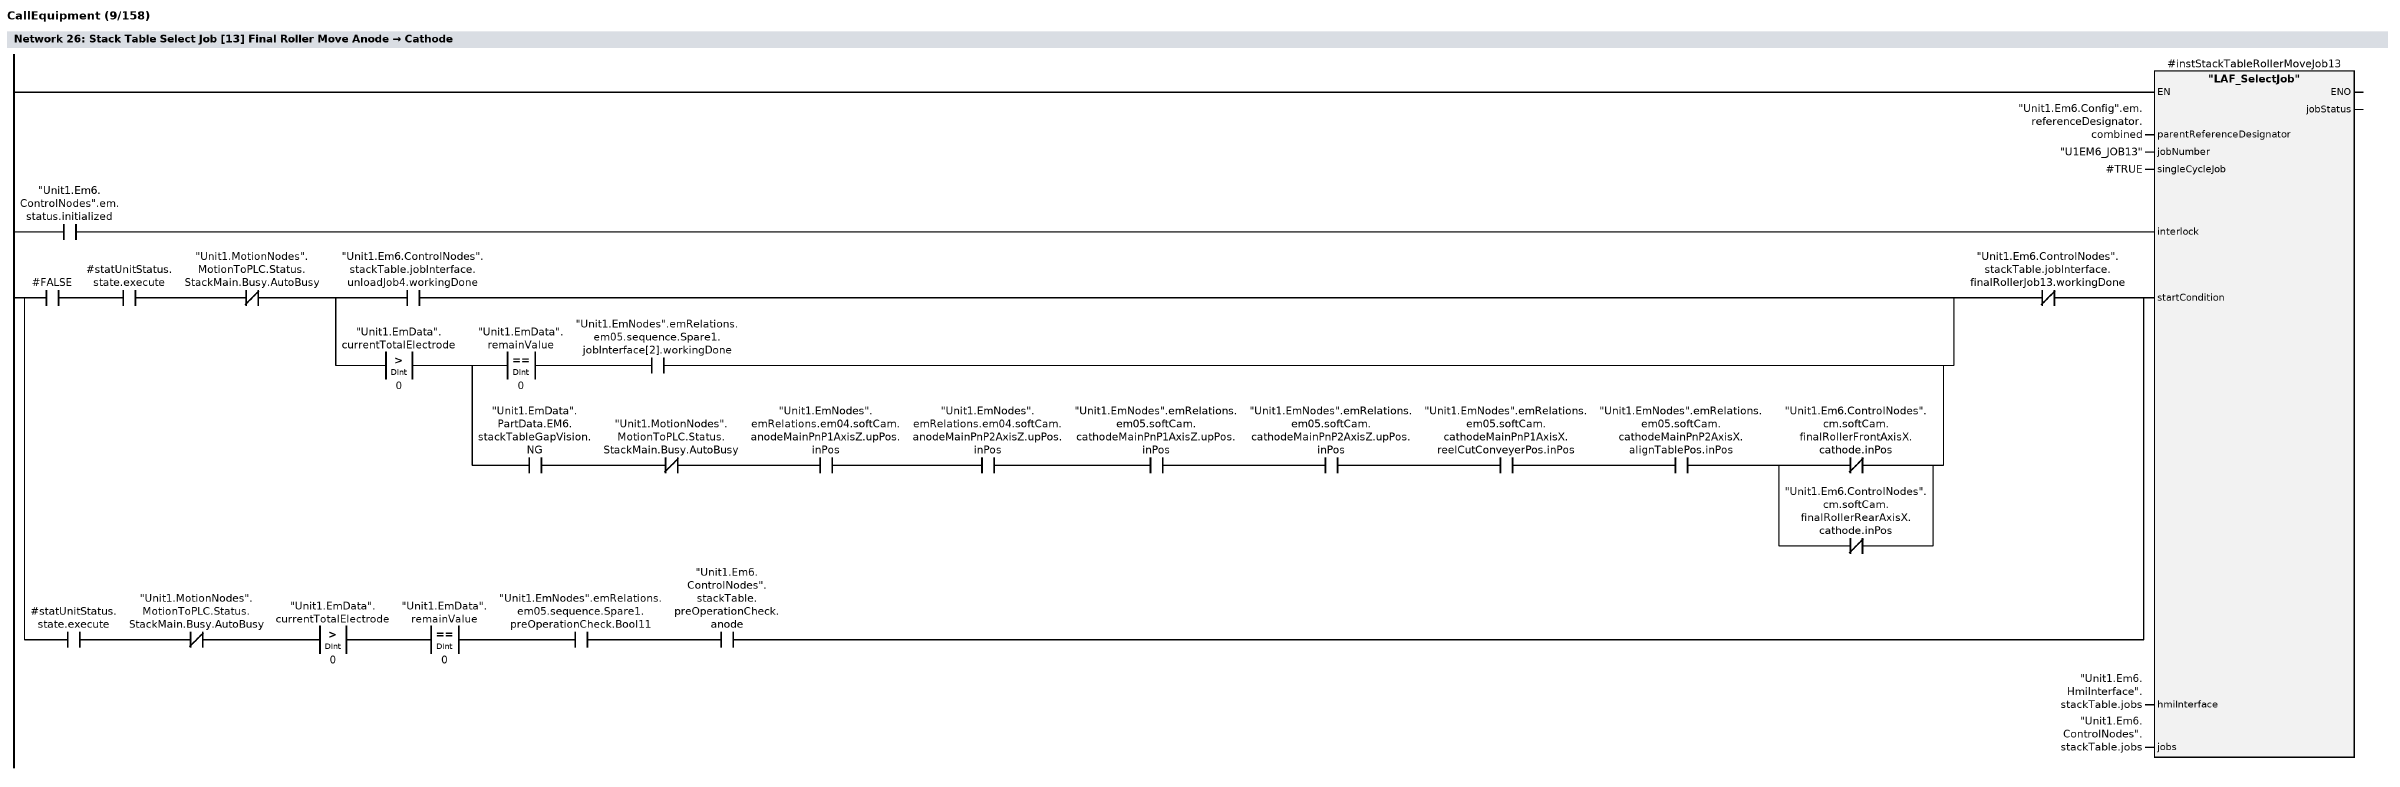
   RUNG wire#powerrail
      #instStackTableRollerMoveJob13(interlock := wire#w1, startCondition := wire#w6, parentReferenceDesignator := "Unit1.Em6.Config".em.referenceDesignator.combined, jobNumber := "U1EM6_JOB13", singleCycleJob := #TRUE, hmiInterface := "Unit1.Em6.HmiInterface".stackTable.jobs, jobs := "Unit1.Em6.ControlNodes".stackTable.jobs, jobStatus =>)
   END_RUNG
   RUNG wire#powerrail
      Contact( "Unit1.Em6.ControlNodes".em.status.initialized )
   END_RUNG wire#w1
   RUNG wire#powerrail
      Contact( #FALSE )
      Contact( #statUnitStatus.state.execute )
      I_Contact( "Unit1.MotionNodes".MotionToPLC.Status.StackMain.Busy.AutoBusy )
      wire#w2
      Contact( "Unit1.Em6.ControlNodes".stackTable.jobInterface.unloadJob4.workingDone )
      wire#w3
      I_Contact( "Unit1.Em6.ControlNodes".stackTable.jobInterface.finalRollerJob13.workingDone )
   END_RUNG wire#w6
   RUNG wire#w2
      { S7_Templates := "SrcType := DInt" } GT_Contact(in1 := "Unit1.EmData".currentTotalElectrode, in2 := 0)
      wire#w4
      { S7_Templates := "SrcType := DInt" } EQ_Contact(in1 := "Unit1.EmData".remainValue, in2 := 0)
      Contact( "Unit1.EmNodes".emRelations.em05.sequence.Spare1.jobInterface[2].workingDone )
   END_RUNG wire#w3
   RUNG wire#w4
      Contact( "Unit1.EmData".PartData.EM6.stackTableGapVision.NG )
      I_Contact( "Unit1.MotionNodes".MotionToPLC.Status.StackMain.Busy.AutoBusy )
      Contact( "Unit1.EmNodes".emRelations.em04.softCam.anodeMainPnP1AxisZ.upPos.inPos )
      Contact( "Unit1.EmNodes".emRelations.em04.softCam.anodeMainPnP2AxisZ.upPos.inPos )
      Contact( "Unit1.EmNodes".emRelations.em05.softCam.cathodeMainPnP1AxisZ.upPos.inPos )
      Contact( "Unit1.EmNodes".emRelations.em05.softCam.cathodeMainPnP2AxisZ.upPos.inPos )
      Contact( "Unit1.EmNodes".emRelations.em05.softCam.cathodeMainPnP1AxisX.reelCutConveyerPos.inPos )
      Contact( "Unit1.EmNodes".emRelations.em05.softCam.cathodeMainPnP2AxisX.alignTablePos.inPos )
      wire#w5
      I_Contact( "Unit1.Em6.ControlNodes".cm.softCam.finalRollerFrontAxisX.cathode.inPos )
   END_RUNG wire#w3
   RUNG wire#w5
      I_Contact( "Unit1.Em6.ControlNodes".cm.softCam.finalRollerRearAxisX.cathode.inPos )
   END_RUNG wire#w3
   RUNG wire#powerrail
      Contact( #statUnitStatus.state.execute )
      I_Contact( "Unit1.MotionNodes".MotionToPLC.Status.StackMain.Busy.AutoBusy )
      { S7_Templates := "SrcType := DInt" } GT_Contact(in1 := "Unit1.EmData".currentTotalElectrode, in2 := 0)
      { S7_Templates := "SrcType := DInt" } EQ_Contact(in1 := "Unit1.EmData".remainValue, in2 := 0)
      Contact( "Unit1.EmNodes".emRelations.em05.sequence.Spare1.preOperationCheck.Bool11 )
      Contact( "Unit1.Em6.ControlNodes".stackTable.preOperationCheck.anode )
   END_RUNG wire#w6
   // the same network as SCL:
   #instStackTableRollerMoveJob13(parentReferenceDesignator := "Unit1.Em6.Config".em.referenceDesignator.combined,   // "LAF_SelectJob"
                           jobNumber := "U1EM6_JOB13",
                           singleCycleJob := #TRUE,
                           interlock := "Unit1.Em6.ControlNodes".em.status.initialized,
                           startCondition := (#FALSE AND #statUnitStatus.state.execute AND NOT "Unit1.MotionNodes".MotionToPLC.Status.StackMain.Busy.AutoBusy AND ("Unit1.Em6.ControlNodes".stackTable.jobInterface.unloadJob4.workingDone OR (("Unit1.EmData".currentTotalElectrode > 0) AND ((("Unit1.EmData".remainValue = 0) AND "Unit1.EmNodes".emRelations.em05.sequence.Spare1.jobInterface[2].workingDone) OR ("Unit1.EmData".PartData.EM6.stackTableGapVision.NG AND NOT "Unit1.MotionNodes".MotionToPLC.Status.StackMain.Busy.AutoBusy AND "Unit1.EmNodes".emRelations.em04.softCam.anodeMainPnP1AxisZ.upPos.inPos AND "Unit1.EmNodes".emRelations.em04.softCam.anodeMainPnP2AxisZ.upPos.inPos AND "Unit1.EmNodes".emRelations.em05.softCam.cathodeMainPnP1AxisZ.upPos.inPos AND "Unit1.EmNodes".emRelations.em05.softCam.cathodeMainPnP2AxisZ.upPos.inPos AND "Unit1.EmNodes".emRelations.em05.softCam.cathodeMainPnP1AxisX.reelCutConveyerPos.inPos AND "Unit1.EmNodes".emRelations.em05.softCam.cathodeMainPnP2AxisX.alignTablePos.inPos AND (NOT "Unit1.Em6.ControlNodes".cm.softCam.finalRollerFrontAxisX.cathode.inPos OR NOT "Unit1.Em6.ControlNodes".cm.softCam.finalRollerRearAxisX.cathode.inPos))))) AND NOT "Unit1.Em6.ControlNodes".stackTable.jobInterface.finalRollerJob13.workingDone) OR (#statUnitStatus.state.execute AND NOT "Unit1.MotionNodes".MotionToPLC.Status.StackMain.Busy.AutoBusy AND ("Unit1.EmData".currentTotalElectrode > 0) AND ("Unit1.EmData".remainValue = 0) AND "Unit1.EmNodes".emRelations.em05.sequence.Spare1.preOperationCheck.Bool11 AND "Unit1.Em6.ControlNodes".stackTable.preOperationCheck.anode),
                           hmiInterface := "Unit1.Em6.HmiInterface".stackTable.jobs,
                           jobs := "Unit1.Em6.ControlNodes".stackTable.jobs);
END_REGION

REGION Network 27: Stack Table Select Job [22] Anode Mendrel
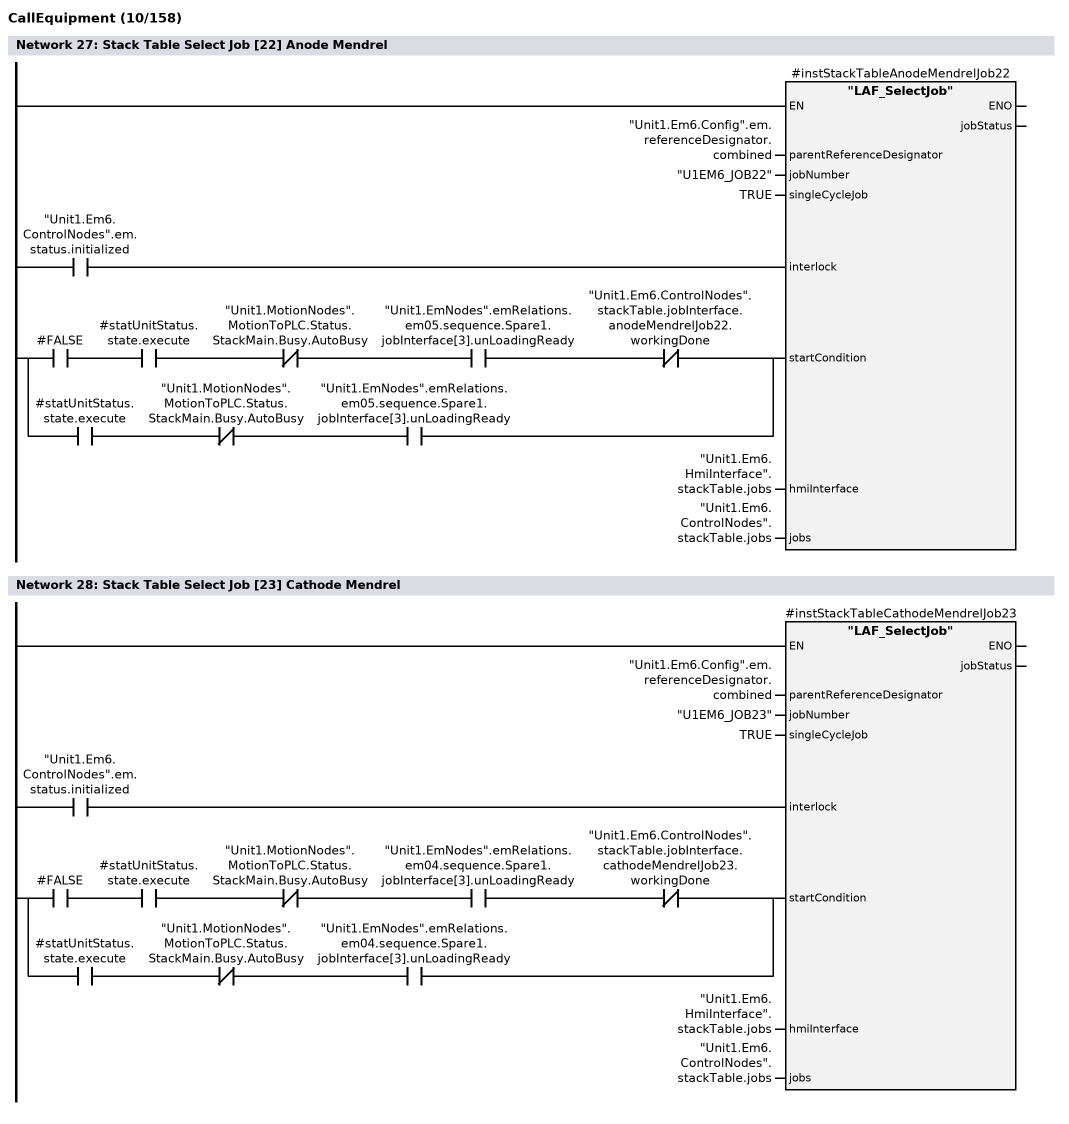
   RUNG wire#powerrail
      #instStackTableAnodeMendrelJob22(interlock := wire#w1, startCondition := wire#w2, parentReferenceDesignator := "Unit1.Em6.Config".em.referenceDesignator.combined, jobNumber := "U1EM6_JOB22", singleCycleJob := TRUE, hmiInterface := "Unit1.Em6.HmiInterface".stackTable.jobs, jobs := "Unit1.Em6.ControlNodes".stackTable.jobs, jobStatus =>)
   END_RUNG
   RUNG wire#powerrail
      Contact( "Unit1.Em6.ControlNodes".em.status.initialized )
   END_RUNG wire#w1
   RUNG wire#powerrail
      Contact( #FALSE )
      Contact( #statUnitStatus.state.execute )
      I_Contact( "Unit1.MotionNodes".MotionToPLC.Status.StackMain.Busy.AutoBusy )
      Contact( "Unit1.EmNodes".emRelations.em05.sequence.Spare1.jobInterface[3].unLoadingReady )
      I_Contact( "Unit1.Em6.ControlNodes".stackTable.jobInterface.anodeMendrelJob22.workingDone )
   END_RUNG wire#w2
   RUNG wire#powerrail
      Contact( #statUnitStatus.state.execute )
      I_Contact( "Unit1.MotionNodes".MotionToPLC.Status.StackMain.Busy.AutoBusy )
      Contact( "Unit1.EmNodes".emRelations.em05.sequence.Spare1.jobInterface[3].unLoadingReady )
   END_RUNG wire#w2
   // the same network as SCL:
   #instStackTableAnodeMendrelJob22(parentReferenceDesignator := "Unit1.Em6.Config".em.referenceDesignator.combined,   // "LAF_SelectJob"
                           jobNumber := "U1EM6_JOB22",
                           singleCycleJob := TRUE,
                           interlock := "Unit1.Em6.ControlNodes".em.status.initialized,
                           startCondition := (#FALSE AND #statUnitStatus.state.execute AND NOT "Unit1.MotionNodes".MotionToPLC.Status.StackMain.Busy.AutoBusy AND "Unit1.EmNodes".emRelations.em05.sequence.Spare1.jobInterface[3].unLoadingReady AND NOT "Unit1.Em6.ControlNodes".stackTable.jobInterface.anodeMendrelJob22.workingDone) OR (#statUnitStatus.state.execute AND NOT "Unit1.MotionNodes".MotionToPLC.Status.StackMain.Busy.AutoBusy AND "Unit1.EmNodes".emRelations.em05.sequence.Spare1.jobInterface[3].unLoadingReady),
                           hmiInterface := "Unit1.Em6.HmiInterface".stackTable.jobs,
                           jobs := "Unit1.Em6.ControlNodes".stackTable.jobs);
END_REGION

REGION Network 28: Stack Table Select Job [23] Cathode Mendrel
   RUNG wire#powerrail
      #instStackTableCathodeMendrelJob23(interlock := wire#w1, startCondition := wire#w2, parentReferenceDesignator := "Unit1.Em6.Config".em.referenceDesignator.combined, jobNumber := "U1EM6_JOB23", singleCycleJob := TRUE, hmiInterface := "Unit1.Em6.HmiInterface".stackTable.jobs, jobs := "Unit1.Em6.ControlNodes".stackTable.jobs, jobStatus =>)
   END_RUNG
   RUNG wire#powerrail
      Contact( "Unit1.Em6.ControlNodes".em.status.initialized )
   END_RUNG wire#w1
   RUNG wire#powerrail
      Contact( #FALSE )
      Contact( #statUnitStatus.state.execute )
      I_Contact( "Unit1.MotionNodes".MotionToPLC.Status.StackMain.Busy.AutoBusy )
      Contact( "Unit1.EmNodes".emRelations.em04.sequence.Spare1.jobInterface[3].unLoadingReady )
      I_Contact( "Unit1.Em6.ControlNodes".stackTable.jobInterface.cathodeMendrelJob23.workingDone )
   END_RUNG wire#w2
   RUNG wire#powerrail
      Contact( #statUnitStatus.state.execute )
      I_Contact( "Unit1.MotionNodes".MotionToPLC.Status.StackMain.Busy.AutoBusy )
      Contact( "Unit1.EmNodes".emRelations.em04.sequence.Spare1.jobInterface[3].unLoadingReady )
   END_RUNG wire#w2
   // the same network as SCL:
   #instStackTableCathodeMendrelJob23(parentReferenceDesignator := "Unit1.Em6.Config".em.referenceDesignator.combined,   // "LAF_SelectJob"
                           jobNumber := "U1EM6_JOB23",
                           singleCycleJob := TRUE,
                           interlock := "Unit1.Em6.ControlNodes".em.status.initialized,
                           startCondition := (#FALSE AND #statUnitStatus.state.execute AND NOT "Unit1.MotionNodes".MotionToPLC.Status.StackMain.Busy.AutoBusy AND "Unit1.EmNodes".emRelations.em04.sequence.Spare1.jobInterface[3].unLoadingReady AND NOT "Unit1.Em6.ControlNodes".stackTable.jobInterface.cathodeMendrelJob23.workingDone) OR (#statUnitStatus.state.execute AND NOT "Unit1.MotionNodes".MotionToPLC.Status.StackMain.Busy.AutoBusy AND "Unit1.EmNodes".emRelations.em04.sequence.Spare1.jobInterface[3].unLoadingReady),
                           hmiInterface := "Unit1.Em6.HmiInterface".stackTable.jobs,
                           jobs := "Unit1.Em6.ControlNodes".stackTable.jobs);
END_REGION

REGION Network 29: Stack Table Select Job [30] Vision
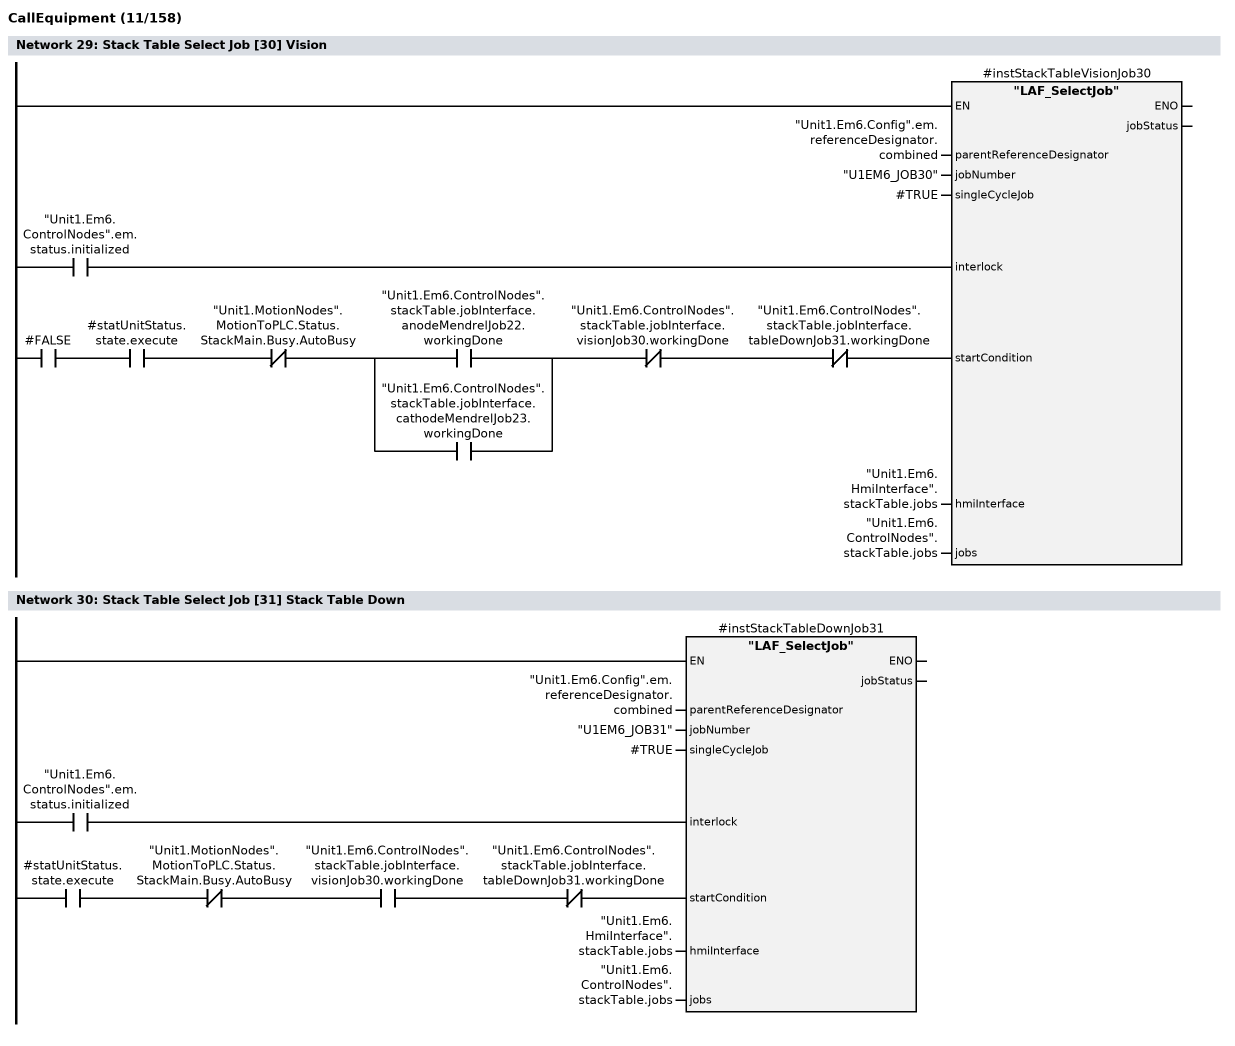
   RUNG wire#powerrail
      #instStackTableVisionJob30(interlock := wire#w1, startCondition := wire#w4, parentReferenceDesignator := "Unit1.Em6.Config".em.referenceDesignator.combined, jobNumber := "U1EM6_JOB30", singleCycleJob := #TRUE, hmiInterface := "Unit1.Em6.HmiInterface".stackTable.jobs, jobs := "Unit1.Em6.ControlNodes".stackTable.jobs, jobStatus =>)
   END_RUNG
   RUNG wire#powerrail
      Contact( "Unit1.Em6.ControlNodes".em.status.initialized )
   END_RUNG wire#w1
   RUNG wire#powerrail
      Contact( #FALSE )
      Contact( #statUnitStatus.state.execute )
      I_Contact( "Unit1.MotionNodes".MotionToPLC.Status.StackMain.Busy.AutoBusy )
      wire#w2
      Contact( "Unit1.Em6.ControlNodes".stackTable.jobInterface.anodeMendrelJob22.workingDone )
      wire#w3
      I_Contact( "Unit1.Em6.ControlNodes".stackTable.jobInterface.visionJob30.workingDone )
      I_Contact( "Unit1.Em6.ControlNodes".stackTable.jobInterface.tableDownJob31.workingDone )
   END_RUNG wire#w4
   RUNG wire#w2
      Contact( "Unit1.Em6.ControlNodes".stackTable.jobInterface.cathodeMendrelJob23.workingDone )
   END_RUNG wire#w3
   // the same network as SCL:
   #instStackTableVisionJob30(parentReferenceDesignator := "Unit1.Em6.Config".em.referenceDesignator.combined,   // "LAF_SelectJob"
                           jobNumber := "U1EM6_JOB30",
                           singleCycleJob := #TRUE,
                           interlock := "Unit1.Em6.ControlNodes".em.status.initialized,
                           startCondition := #FALSE AND #statUnitStatus.state.execute AND NOT "Unit1.MotionNodes".MotionToPLC.Status.StackMain.Busy.AutoBusy AND ("Unit1.Em6.ControlNodes".stackTable.jobInterface.anodeMendrelJob22.workingDone OR "Unit1.Em6.ControlNodes".stackTable.jobInterface.cathodeMendrelJob23.workingDone) AND NOT "Unit1.Em6.ControlNodes".stackTable.jobInterface.visionJob30.workingDone AND NOT "Unit1.Em6.ControlNodes".stackTable.jobInterface.tableDownJob31.workingDone,
                           hmiInterface := "Unit1.Em6.HmiInterface".stackTable.jobs,
                           jobs := "Unit1.Em6.ControlNodes".stackTable.jobs);
END_REGION

REGION Network 30: Stack Table Select Job [31] Stack Table Down
   RUNG wire#powerrail
      #instStackTableDownJob31(interlock := wire#w1, startCondition := wire#w2, parentReferenceDesignator := "Unit1.Em6.Config".em.referenceDesignator.combined, jobNumber := "U1EM6_JOB31", singleCycleJob := #TRUE, hmiInterface := "Unit1.Em6.HmiInterface".stackTable.jobs, jobs := "Unit1.Em6.ControlNodes".stackTable.jobs, jobStatus =>)
   END_RUNG
   RUNG wire#powerrail
      Contact( "Unit1.Em6.ControlNodes".em.status.initialized )
   END_RUNG wire#w1
   RUNG wire#powerrail
      Contact( #statUnitStatus.state.execute )
      I_Contact( "Unit1.MotionNodes".MotionToPLC.Status.StackMain.Busy.AutoBusy )
      Contact( "Unit1.Em6.ControlNodes".stackTable.jobInterface.visionJob30.workingDone )
      I_Contact( "Unit1.Em6.ControlNodes".stackTable.jobInterface.tableDownJob31.workingDone )
   END_RUNG wire#w2
   // the same network as SCL:
   #instStackTableDownJob31(parentReferenceDesignator := "Unit1.Em6.Config".em.referenceDesignator.combined,   // "LAF_SelectJob"
                           jobNumber := "U1EM6_JOB31",
                           singleCycleJob := #TRUE,
                           interlock := "Unit1.Em6.ControlNodes".em.status.initialized,
                           startCondition := #statUnitStatus.state.execute AND NOT "Unit1.MotionNodes".MotionToPLC.Status.StackMain.Busy.AutoBusy AND "Unit1.Em6.ControlNodes".stackTable.jobInterface.visionJob30.workingDone AND NOT "Unit1.Em6.ControlNodes".stackTable.jobInterface.tableDownJob31.workingDone,
                           hmiInterface := "Unit1.Em6.HmiInterface".stackTable.jobs,
                           jobs := "Unit1.Em6.ControlNodes".stackTable.jobs);
END_REGION

REGION Network 31: Stack Table Select Job [04] Unload
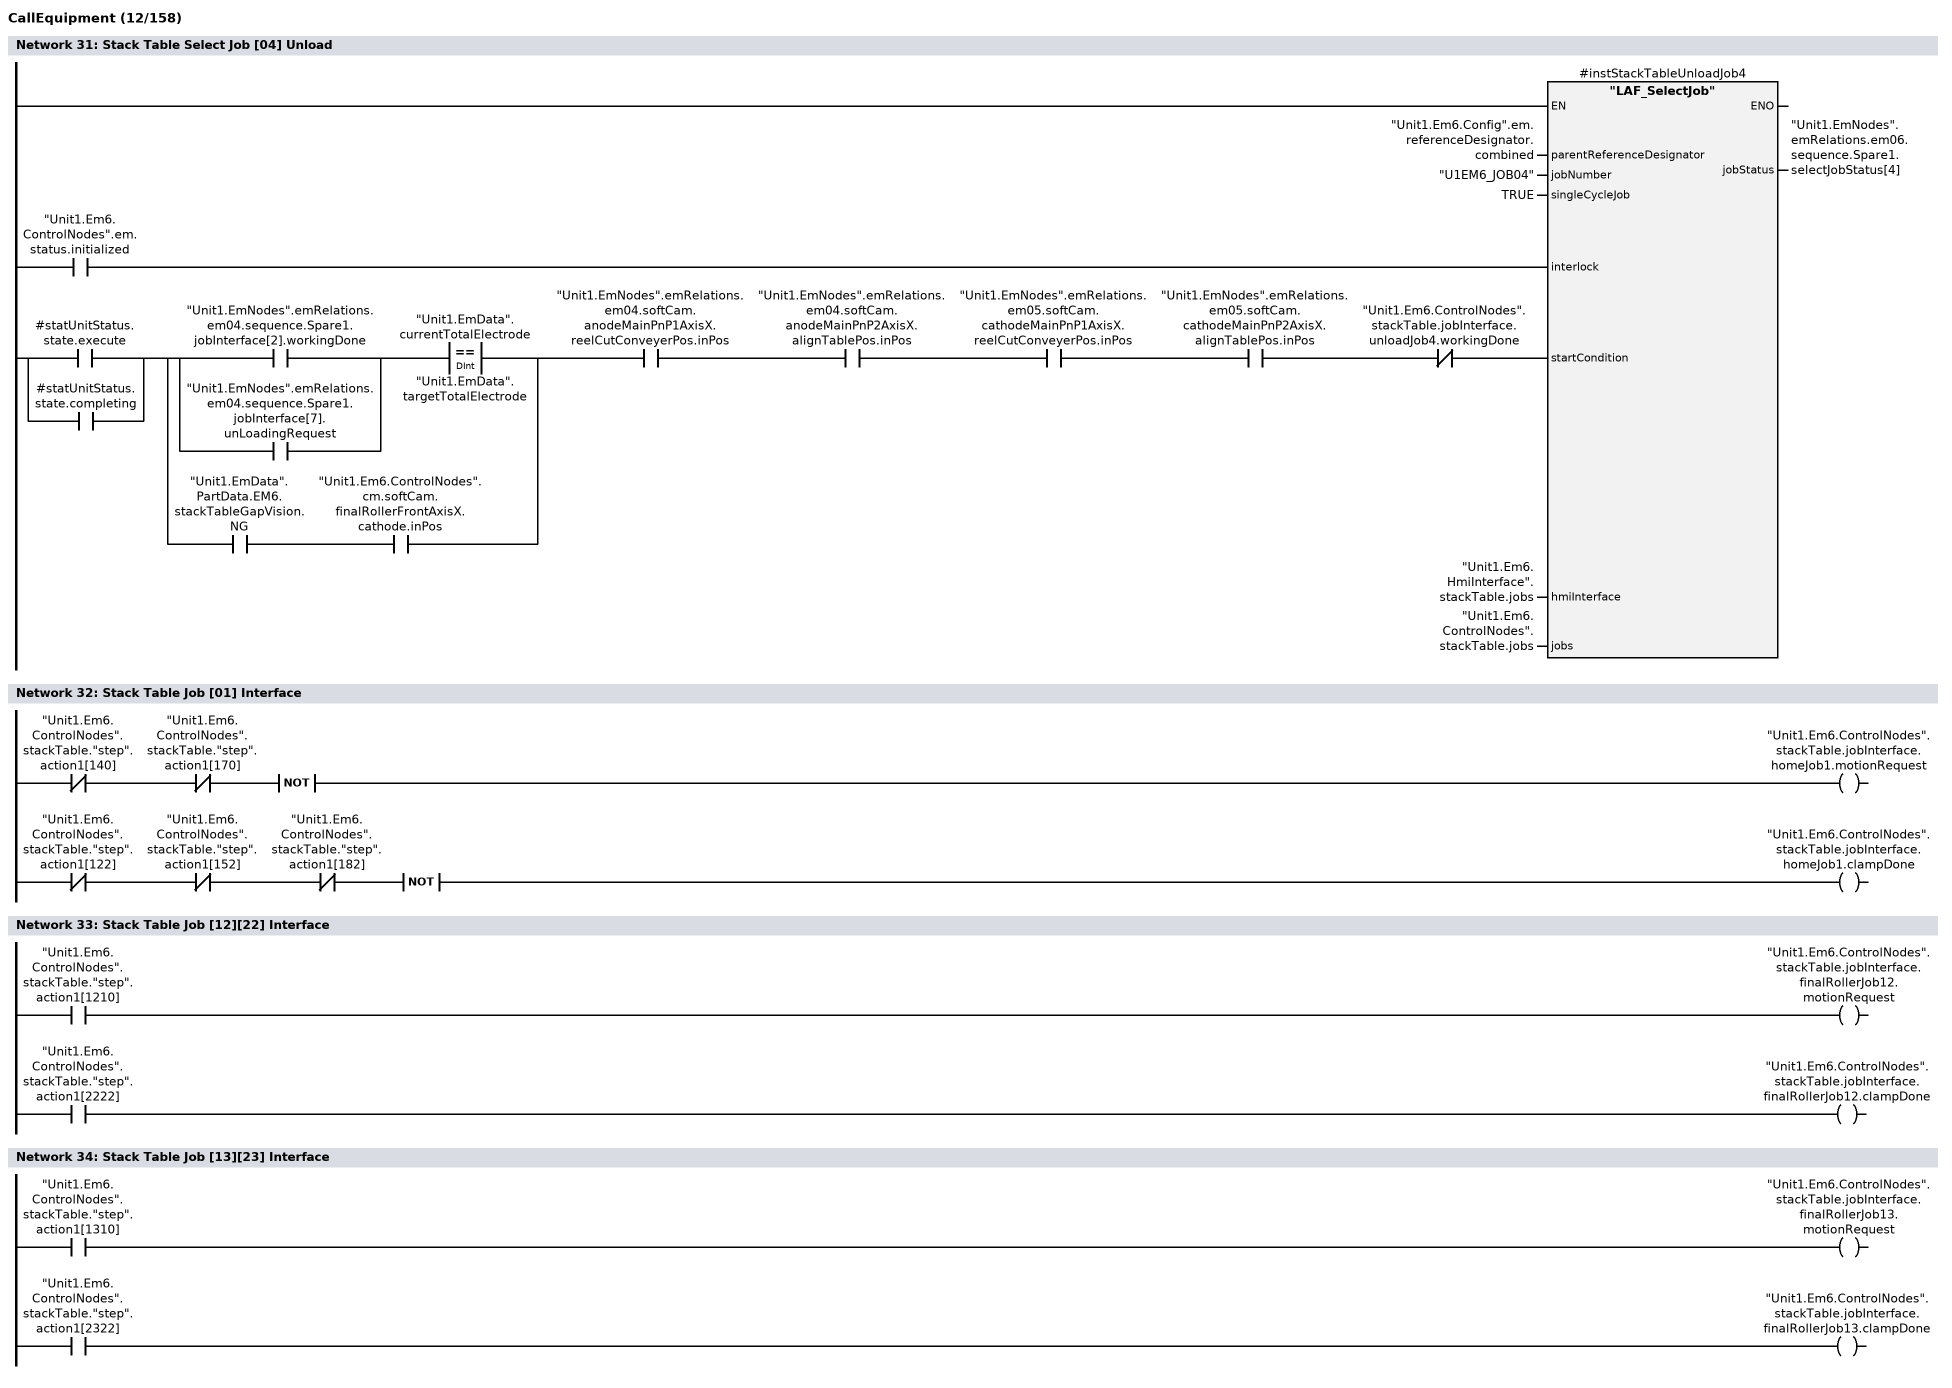
   RUNG wire#powerrail
      #instStackTableUnloadJob4(interlock := wire#w1, startCondition := wire#w5, parentReferenceDesignator := "Unit1.Em6.Config".em.referenceDesignator.combined, jobNumber := "U1EM6_JOB04", singleCycleJob := TRUE, hmiInterface := "Unit1.Em6.HmiInterface".stackTable.jobs, jobs := "Unit1.Em6.ControlNodes".stackTable.jobs, jobStatus => "Unit1.EmNodes".emRelations.em06.sequence.Spare1.selectJobStatus[4])
   END_RUNG
   RUNG wire#powerrail
      Contact( "Unit1.Em6.ControlNodes".em.status.initialized )
   END_RUNG wire#w1
   RUNG wire#powerrail
      Contact( #statUnitStatus.state.execute )
      wire#w2
      Contact( "Unit1.EmNodes".emRelations.em04.sequence.Spare1.jobInterface[2].workingDone )
      wire#w3
      { S7_Templates := "SrcType := DInt" } EQ_Contact(in1 := "Unit1.EmData".currentTotalElectrode, in2 := "Unit1.EmData".targetTotalElectrode)
      wire#w4
      Contact( "Unit1.EmNodes".emRelations.em04.softCam.anodeMainPnP1AxisX.reelCutConveyerPos.inPos )
      Contact( "Unit1.EmNodes".emRelations.em04.softCam.anodeMainPnP2AxisX.alignTablePos.inPos )
      Contact( "Unit1.EmNodes".emRelations.em05.softCam.cathodeMainPnP1AxisX.reelCutConveyerPos.inPos )
      Contact( "Unit1.EmNodes".emRelations.em05.softCam.cathodeMainPnP2AxisX.alignTablePos.inPos )
      I_Contact( "Unit1.Em6.ControlNodes".stackTable.jobInterface.unloadJob4.workingDone )
   END_RUNG wire#w5
   RUNG wire#powerrail
      Contact( #statUnitStatus.state.completing )
   END_RUNG wire#w2
   RUNG wire#w2
      Contact( "Unit1.EmNodes".emRelations.em04.sequence.Spare1.jobInterface[7].unLoadingRequest )
   END_RUNG wire#w3
   RUNG wire#w2
      Contact( "Unit1.EmData".PartData.EM6.stackTableGapVision.NG )
      Contact( "Unit1.Em6.ControlNodes".cm.softCam.finalRollerFrontAxisX.cathode.inPos )
   END_RUNG wire#w4
   // the same network as SCL:
   #instStackTableUnloadJob4(parentReferenceDesignator := "Unit1.Em6.Config".em.referenceDesignator.combined,   // "LAF_SelectJob"
                           jobNumber := "U1EM6_JOB04",
                           singleCycleJob := TRUE,
                           interlock := "Unit1.Em6.ControlNodes".em.status.initialized,
                           startCondition := (#statUnitStatus.state.execute OR #statUnitStatus.state.completing) AND ((("Unit1.EmNodes".emRelations.em04.sequence.Spare1.jobInterface[2].workingDone OR "Unit1.EmNodes".emRelations.em04.sequence.Spare1.jobInterface[7].unLoadingRequest) AND ("Unit1.EmData".currentTotalElectrode = "Unit1.EmData".targetTotalElectrode)) OR ("Unit1.EmData".PartData.EM6.stackTableGapVision.NG AND "Unit1.Em6.ControlNodes".cm.softCam.finalRollerFrontAxisX.cathode.inPos)) AND "Unit1.EmNodes".emRelations.em04.softCam.anodeMainPnP1AxisX.reelCutConveyerPos.inPos AND "Unit1.EmNodes".emRelations.em04.softCam.anodeMainPnP2AxisX.alignTablePos.inPos AND "Unit1.EmNodes".emRelations.em05.softCam.cathodeMainPnP1AxisX.reelCutConveyerPos.inPos AND "Unit1.EmNodes".emRelations.em05.softCam.cathodeMainPnP2AxisX.alignTablePos.inPos AND NOT "Unit1.Em6.ControlNodes".stackTable.jobInterface.unloadJob4.workingDone,
                           hmiInterface := "Unit1.Em6.HmiInterface".stackTable.jobs,
                           jobs := "Unit1.Em6.ControlNodes".stackTable.jobs,
                           jobStatus => "Unit1.EmNodes".emRelations.em06.sequence.Spare1.selectJobStatus[4]);
END_REGION

REGION Network 32: Stack Table Job [01] Interface
   RUNG wire#powerrail
      I_Contact( "Unit1.Em6.ControlNodes".stackTable."step".action1[140] )
      I_Contact( "Unit1.Em6.ControlNodes".stackTable."step".action1[170] )
      Not()
      Coil( "Unit1.Em6.ControlNodes".stackTable.jobInterface.homeJob1.motionRequest )
   END_RUNG
   RUNG wire#powerrail
      I_Contact( "Unit1.Em6.ControlNodes".stackTable."step".action1[122] )
      I_Contact( "Unit1.Em6.ControlNodes".stackTable."step".action1[152] )
      I_Contact( "Unit1.Em6.ControlNodes".stackTable."step".action1[182] )
      Not()
      Coil( "Unit1.Em6.ControlNodes".stackTable.jobInterface.homeJob1.clampDone )
   END_RUNG
   // the same network as SCL:
   "Unit1.Em6.ControlNodes".stackTable.jobInterface.homeJob1.motionRequest := NOT (NOT "Unit1.Em6.ControlNodes".stackTable."step".action1[140] AND NOT "Unit1.Em6.ControlNodes".stackTable."step".action1[170]);
   "Unit1.Em6.ControlNodes".stackTable.jobInterface.homeJob1.clampDone := NOT (NOT "Unit1.Em6.ControlNodes".stackTable."step".action1[122] AND NOT "Unit1.Em6.ControlNodes".stackTable."step".action1[152] AND NOT "Unit1.Em6.ControlNodes".stackTable."step".action1[182]);
END_REGION

REGION Network 33: Stack Table Job [12][22] Interface
   RUNG wire#powerrail
      Contact( "Unit1.Em6.ControlNodes".stackTable."step".action1[1210] )
      Coil( "Unit1.Em6.ControlNodes".stackTable.jobInterface.finalRollerJob12.motionRequest )
   END_RUNG
   RUNG wire#powerrail
      Contact( "Unit1.Em6.ControlNodes".stackTable."step".action1[2222] )
      Coil( "Unit1.Em6.ControlNodes".stackTable.jobInterface.finalRollerJob12.clampDone )
   END_RUNG
   // the same network as SCL:
   "Unit1.Em6.ControlNodes".stackTable.jobInterface.finalRollerJob12.motionRequest := "Unit1.Em6.ControlNodes".stackTable."step".action1[1210];
   "Unit1.Em6.ControlNodes".stackTable.jobInterface.finalRollerJob12.clampDone := "Unit1.Em6.ControlNodes".stackTable."step".action1[2222];
END_REGION

REGION Network 34: Stack Table Job [13][23] Interface
   RUNG wire#powerrail
      Contact( "Unit1.Em6.ControlNodes".stackTable."step".action1[1310] )
      Coil( "Unit1.Em6.ControlNodes".stackTable.jobInterface.finalRollerJob13.motionRequest )
   END_RUNG
   RUNG wire#powerrail
      Contact( "Unit1.Em6.ControlNodes".stackTable."step".action1[2322] )
      Coil( "Unit1.Em6.ControlNodes".stackTable.jobInterface.finalRollerJob13.clampDone )
   END_RUNG
   // the same network as SCL:
   "Unit1.Em6.ControlNodes".stackTable.jobInterface.finalRollerJob13.motionRequest := "Unit1.Em6.ControlNodes".stackTable."step".action1[1310];
   "Unit1.Em6.ControlNodes".stackTable.jobInterface.finalRollerJob13.clampDone := "Unit1.Em6.ControlNodes".stackTable."step".action1[2322];
END_REGION

REGION Network 35: Stack Table Job [04] Interface
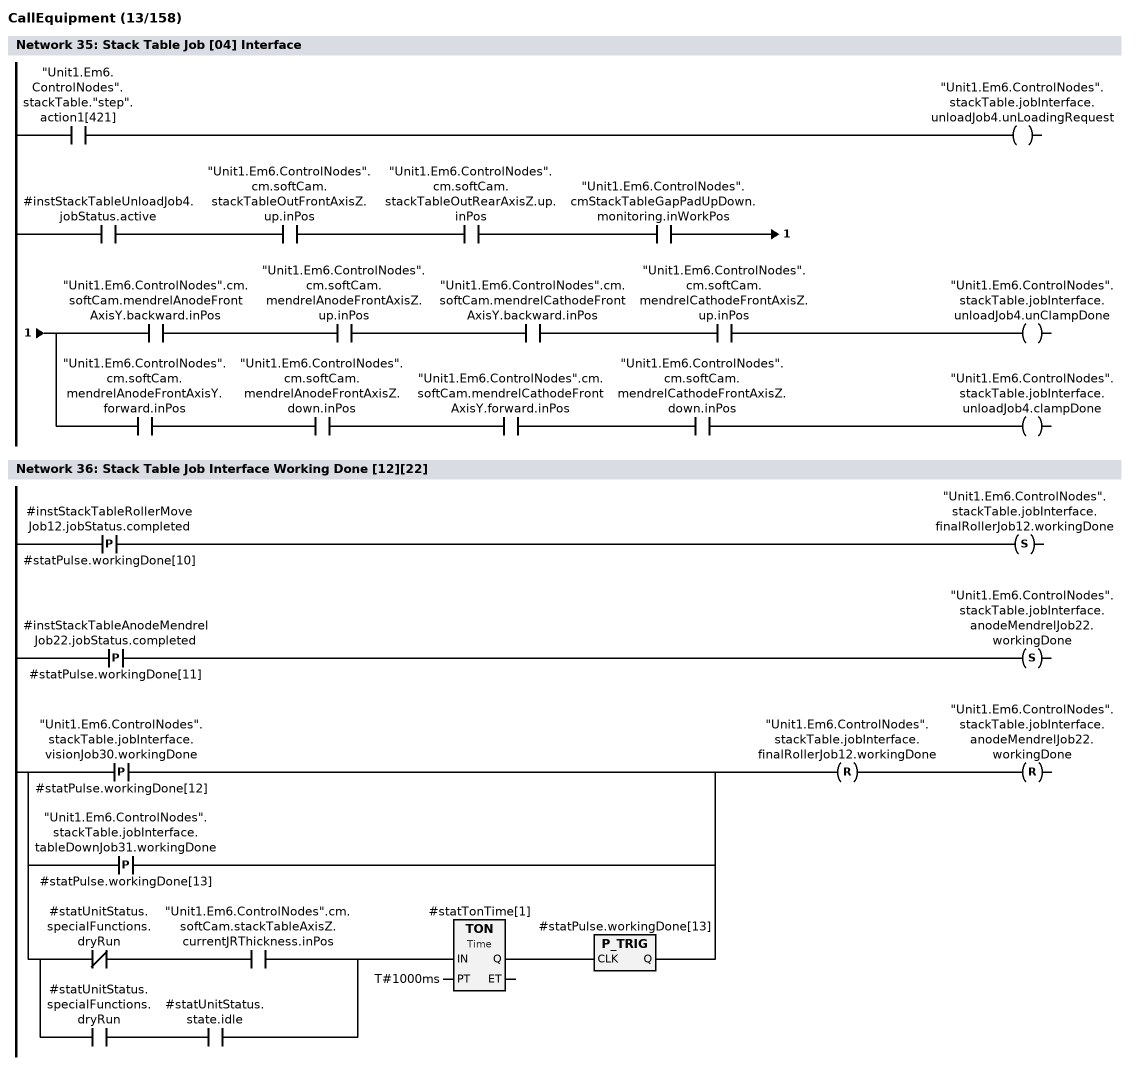
   RUNG wire#powerrail
      Contact( "Unit1.Em6.ControlNodes".stackTable."step".action1[421] )
      Coil( "Unit1.Em6.ControlNodes".stackTable.jobInterface.unloadJob4.unLoadingRequest )
   END_RUNG
   RUNG wire#powerrail
      Contact( #instStackTableUnloadJob4.jobStatus.active )
      Contact( "Unit1.Em6.ControlNodes".cm.softCam.stackTableOutFrontAxisZ.up.inPos )
      Contact( "Unit1.Em6.ControlNodes".cm.softCam.stackTableOutRearAxisZ.up.inPos )
      Contact( "Unit1.Em6.ControlNodes".cmStackTableGapPadUpDown.monitoring.inWorkPos )
      wire#w1
      Contact( "Unit1.Em6.ControlNodes".cm.softCam.mendrelAnodeFrontAxisY.backward.inPos )
      Contact( "Unit1.Em6.ControlNodes".cm.softCam.mendrelAnodeFrontAxisZ.up.inPos )
      Contact( "Unit1.Em6.ControlNodes".cm.softCam.mendrelCathodeFrontAxisY.backward.inPos )
      Contact( "Unit1.Em6.ControlNodes".cm.softCam.mendrelCathodeFrontAxisZ.up.inPos )
      Coil( "Unit1.Em6.ControlNodes".stackTable.jobInterface.unloadJob4.unClampDone )
   END_RUNG
   RUNG wire#w1
      Contact( "Unit1.Em6.ControlNodes".cm.softCam.mendrelAnodeFrontAxisY.forward.inPos )
      Contact( "Unit1.Em6.ControlNodes".cm.softCam.mendrelAnodeFrontAxisZ.down.inPos )
      Contact( "Unit1.Em6.ControlNodes".cm.softCam.mendrelCathodeFrontAxisY.forward.inPos )
      Contact( "Unit1.Em6.ControlNodes".cm.softCam.mendrelCathodeFrontAxisZ.down.inPos )
      Coil( "Unit1.Em6.ControlNodes".stackTable.jobInterface.unloadJob4.clampDone )
   END_RUNG
   // the same network as SCL:
   "Unit1.Em6.ControlNodes".stackTable.jobInterface.unloadJob4.unLoadingRequest := "Unit1.Em6.ControlNodes".stackTable."step".action1[421];
   #_w1 := #instStackTableUnloadJob4.jobStatus.active AND "Unit1.Em6.ControlNodes".cm.softCam.stackTableOutFrontAxisZ.up.inPos AND "Unit1.Em6.ControlNodes".cm.softCam.stackTableOutRearAxisZ.up.inPos AND "Unit1.Em6.ControlNodes".cmStackTableGapPadUpDown.monitoring.inWorkPos;
   "Unit1.Em6.ControlNodes".stackTable.jobInterface.unloadJob4.unClampDone := #_w1 AND "Unit1.Em6.ControlNodes".cm.softCam.mendrelAnodeFrontAxisY.backward.inPos AND "Unit1.Em6.ControlNodes".cm.softCam.mendrelAnodeFrontAxisZ.up.inPos AND "Unit1.Em6.ControlNodes".cm.softCam.mendrelCathodeFrontAxisY.backward.inPos AND "Unit1.Em6.ControlNodes".cm.softCam.mendrelCathodeFrontAxisZ.up.inPos;
   "Unit1.Em6.ControlNodes".stackTable.jobInterface.unloadJob4.clampDone := #_w1 AND "Unit1.Em6.ControlNodes".cm.softCam.mendrelAnodeFrontAxisY.forward.inPos AND "Unit1.Em6.ControlNodes".cm.softCam.mendrelAnodeFrontAxisZ.down.inPos AND "Unit1.Em6.ControlNodes".cm.softCam.mendrelCathodeFrontAxisY.forward.inPos AND "Unit1.Em6.ControlNodes".cm.softCam.mendrelCathodeFrontAxisZ.down.inPos;
END_REGION

REGION Network 36: Stack Table Job Interface Working Done [12][22]
   RUNG wire#powerrail
      P_Contact(operand := #instStackTableRollerMoveJob12.jobStatus.completed, bit := #statPulse.workingDone[10])
      S_Coil( "Unit1.Em6.ControlNodes".stackTable.jobInterface.finalRollerJob12.workingDone )
   END_RUNG
   RUNG wire#powerrail
      P_Contact(operand := #instStackTableAnodeMendrelJob22.jobStatus.completed, bit := #statPulse.workingDone[11])
      S_Coil( "Unit1.Em6.ControlNodes".stackTable.jobInterface.anodeMendrelJob22.workingDone )
   END_RUNG
   RUNG wire#powerrail
      P_Contact(operand := "Unit1.Em6.ControlNodes".stackTable.jobInterface.visionJob30.workingDone, bit := #statPulse.workingDone[12])
      wire#w1
      R_Coil( "Unit1.Em6.ControlNodes".stackTable.jobInterface.finalRollerJob12.workingDone )
      R_Coil( "Unit1.Em6.ControlNodes".stackTable.jobInterface.anodeMendrelJob22.workingDone )
   END_RUNG
   RUNG wire#powerrail
      P_Contact(operand := "Unit1.Em6.ControlNodes".stackTable.jobInterface.tableDownJob31.workingDone, bit := #statPulse.workingDone[13])
   END_RUNG wire#w1
   RUNG wire#powerrail
      I_Contact( #statUnitStatus.specialFunctions.dryRun )
      Contact( "Unit1.Em6.ControlNodes".cm.softCam.stackTableAxisZ.currentJRThickness.inPos )
      wire#w2
      { S7_Templates := "time_type := Time" } #statTonTime[1].TON(pt := T#1000ms, et =>)
      P_Trig( #statPulse.workingDone[13] )
   END_RUNG wire#w1
   RUNG wire#powerrail
      Contact( #statUnitStatus.specialFunctions.dryRun )
      Contact( #statUnitStatus.state.idle )
   END_RUNG wire#w2
   // the same network as SCL:
   #_w1 := #instStackTableRollerMoveJob12.jobStatus.completed AND NOT #statPulse.workingDone[10];   // rising edge of #instStackTableRollerMoveJob12.jobStatus.completed
   #statPulse.workingDone[10] := #instStackTableRollerMoveJob12.jobStatus.completed;
   IF #_w1 THEN
       "Unit1.Em6.ControlNodes".stackTable.jobInterface.finalRollerJob12.workingDone := TRUE;
   END_IF;
   #_w2 := #instStackTableAnodeMendrelJob22.jobStatus.completed AND NOT #statPulse.workingDone[11];   // rising edge of #instStackTableAnodeMendrelJob22.jobStatus.completed
   #statPulse.workingDone[11] := #instStackTableAnodeMendrelJob22.jobStatus.completed;
   IF #_w2 THEN
       "Unit1.Em6.ControlNodes".stackTable.jobInterface.anodeMendrelJob22.workingDone := TRUE;
   END_IF;
   #_w3 := "Unit1.Em6.ControlNodes".stackTable.jobInterface.visionJob30.workingDone AND NOT #statPulse.workingDone[12];   // rising edge of "Unit1.Em6.ControlNodes".stackTable.jobInterface.visionJob30.workingDone
   #statPulse.workingDone[12] := "Unit1.Em6.ControlNodes".stackTable.jobInterface.visionJob30.workingDone;
   #_w4 := "Unit1.Em6.ControlNodes".stackTable.jobInterface.tableDownJob31.workingDone AND NOT #statPulse.workingDone[13];   // rising edge of "Unit1.Em6.ControlNodes".stackTable.jobInterface.tableDownJob31.workingDone
   #statPulse.workingDone[13] := "Unit1.Em6.ControlNodes".stackTable.jobInterface.tableDownJob31.workingDone;
   #statTonTime[1].TON(IN := (NOT #statUnitStatus.specialFunctions.dryRun AND "Unit1.Em6.ControlNodes".cm.softCam.stackTableAxisZ.currentJRThickness.inPos) OR (#statUnitStatus.specialFunctions.dryRun AND #statUnitStatus.state.idle),
                       PT := T#1000ms);
   #_w5 := #statTonTime[1].Q AND NOT #statPulse.workingDone[13];   // rising edge
   #statPulse.workingDone[13] := #statTonTime[1].Q;
   IF #_w3 OR #_w4 OR #_w5 THEN
       "Unit1.Em6.ControlNodes".stackTable.jobInterface.finalRollerJob12.workingDone := FALSE;
       "Unit1.Em6.ControlNodes".stackTable.jobInterface.anodeMendrelJob22.workingDone := FALSE;
   END_IF;
END_REGION

REGION Network 37: Stack Table Job Interface Working Done [13][23]
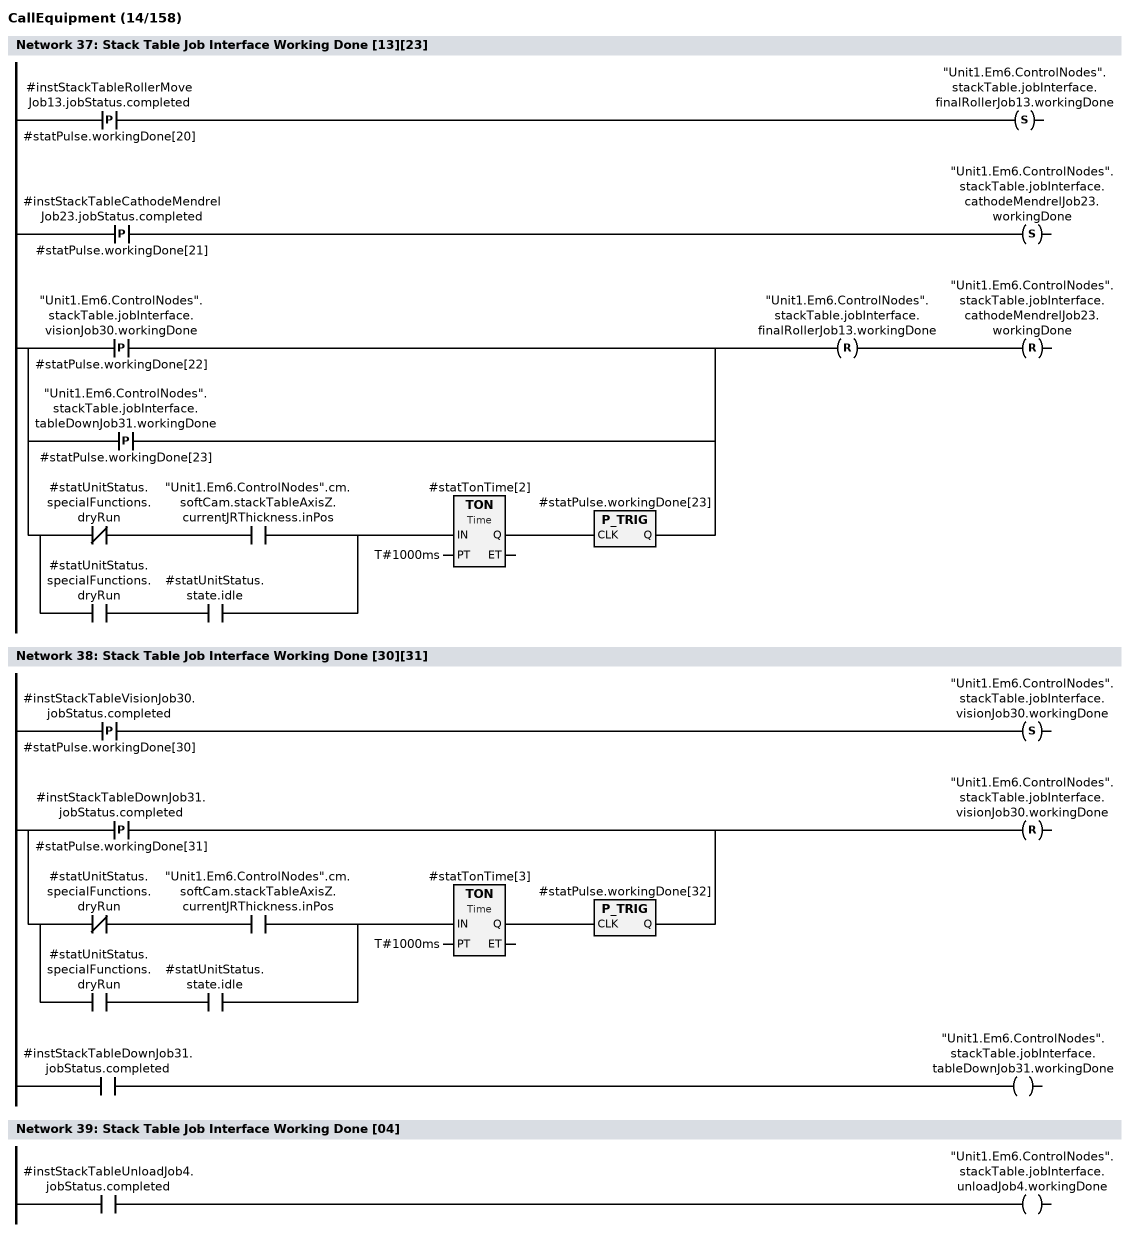
   RUNG wire#powerrail
      P_Contact(operand := #instStackTableRollerMoveJob13.jobStatus.completed, bit := #statPulse.workingDone[20])
      S_Coil( "Unit1.Em6.ControlNodes".stackTable.jobInterface.finalRollerJob13.workingDone )
   END_RUNG
   RUNG wire#powerrail
      P_Contact(operand := #instStackTableCathodeMendrelJob23.jobStatus.completed, bit := #statPulse.workingDone[21])
      S_Coil( "Unit1.Em6.ControlNodes".stackTable.jobInterface.cathodeMendrelJob23.workingDone )
   END_RUNG
   RUNG wire#powerrail
      P_Contact(operand := "Unit1.Em6.ControlNodes".stackTable.jobInterface.visionJob30.workingDone, bit := #statPulse.workingDone[22])
      wire#w1
      R_Coil( "Unit1.Em6.ControlNodes".stackTable.jobInterface.finalRollerJob13.workingDone )
      R_Coil( "Unit1.Em6.ControlNodes".stackTable.jobInterface.cathodeMendrelJob23.workingDone )
   END_RUNG
   RUNG wire#powerrail
      P_Contact(operand := "Unit1.Em6.ControlNodes".stackTable.jobInterface.tableDownJob31.workingDone, bit := #statPulse.workingDone[23])
   END_RUNG wire#w1
   RUNG wire#powerrail
      I_Contact( #statUnitStatus.specialFunctions.dryRun )
      Contact( "Unit1.Em6.ControlNodes".cm.softCam.stackTableAxisZ.currentJRThickness.inPos )
      wire#w2
      { S7_Templates := "time_type := Time" } #statTonTime[2].TON(pt := T#1000ms, et =>)
      P_Trig( #statPulse.workingDone[23] )
   END_RUNG wire#w1
   RUNG wire#powerrail
      Contact( #statUnitStatus.specialFunctions.dryRun )
      Contact( #statUnitStatus.state.idle )
   END_RUNG wire#w2
   // the same network as SCL:
   #_w1 := #instStackTableRollerMoveJob13.jobStatus.completed AND NOT #statPulse.workingDone[20];   // rising edge of #instStackTableRollerMoveJob13.jobStatus.completed
   #statPulse.workingDone[20] := #instStackTableRollerMoveJob13.jobStatus.completed;
   IF #_w1 THEN
       "Unit1.Em6.ControlNodes".stackTable.jobInterface.finalRollerJob13.workingDone := TRUE;
   END_IF;
   #_w2 := #instStackTableCathodeMendrelJob23.jobStatus.completed AND NOT #statPulse.workingDone[21];   // rising edge of #instStackTableCathodeMendrelJob23.jobStatus.completed
   #statPulse.workingDone[21] := #instStackTableCathodeMendrelJob23.jobStatus.completed;
   IF #_w2 THEN
       "Unit1.Em6.ControlNodes".stackTable.jobInterface.cathodeMendrelJob23.workingDone := TRUE;
   END_IF;
   #_w3 := "Unit1.Em6.ControlNodes".stackTable.jobInterface.visionJob30.workingDone AND NOT #statPulse.workingDone[22];   // rising edge of "Unit1.Em6.ControlNodes".stackTable.jobInterface.visionJob30.workingDone
   #statPulse.workingDone[22] := "Unit1.Em6.ControlNodes".stackTable.jobInterface.visionJob30.workingDone;
   #_w4 := "Unit1.Em6.ControlNodes".stackTable.jobInterface.tableDownJob31.workingDone AND NOT #statPulse.workingDone[23];   // rising edge of "Unit1.Em6.ControlNodes".stackTable.jobInterface.tableDownJob31.workingDone
   #statPulse.workingDone[23] := "Unit1.Em6.ControlNodes".stackTable.jobInterface.tableDownJob31.workingDone;
   #statTonTime[2].TON(IN := (NOT #statUnitStatus.specialFunctions.dryRun AND "Unit1.Em6.ControlNodes".cm.softCam.stackTableAxisZ.currentJRThickness.inPos) OR (#statUnitStatus.specialFunctions.dryRun AND #statUnitStatus.state.idle),
                       PT := T#1000ms);
   #_w5 := #statTonTime[2].Q AND NOT #statPulse.workingDone[23];   // rising edge
   #statPulse.workingDone[23] := #statTonTime[2].Q;
   IF #_w3 OR #_w4 OR #_w5 THEN
       "Unit1.Em6.ControlNodes".stackTable.jobInterface.finalRollerJob13.workingDone := FALSE;
       "Unit1.Em6.ControlNodes".stackTable.jobInterface.cathodeMendrelJob23.workingDone := FALSE;
   END_IF;
END_REGION

REGION Network 38: Stack Table Job Interface Working Done [30][31]
   RUNG wire#powerrail
      P_Contact(operand := #instStackTableVisionJob30.jobStatus.completed, bit := #statPulse.workingDone[30])
      S_Coil( "Unit1.Em6.ControlNodes".stackTable.jobInterface.visionJob30.workingDone )
   END_RUNG
   RUNG wire#powerrail
      P_Contact(operand := #instStackTableDownJob31.jobStatus.completed, bit := #statPulse.workingDone[31])
      wire#w1
      R_Coil( "Unit1.Em6.ControlNodes".stackTable.jobInterface.visionJob30.workingDone )
   END_RUNG
   RUNG wire#powerrail
      I_Contact( #statUnitStatus.specialFunctions.dryRun )
      Contact( "Unit1.Em6.ControlNodes".cm.softCam.stackTableAxisZ.currentJRThickness.inPos )
      wire#w2
      { S7_Templates := "time_type := Time" } #statTonTime[3].TON(pt := T#1000ms, et =>)
      P_Trig( #statPulse.workingDone[32] )
   END_RUNG wire#w1
   RUNG wire#powerrail
      Contact( #statUnitStatus.specialFunctions.dryRun )
      Contact( #statUnitStatus.state.idle )
   END_RUNG wire#w2
   RUNG wire#powerrail
      Contact( #instStackTableDownJob31.jobStatus.completed )
      Coil( "Unit1.Em6.ControlNodes".stackTable.jobInterface.tableDownJob31.workingDone )
   END_RUNG
   // the same network as SCL:
   #_w1 := #instStackTableVisionJob30.jobStatus.completed AND NOT #statPulse.workingDone[30];   // rising edge of #instStackTableVisionJob30.jobStatus.completed
   #statPulse.workingDone[30] := #instStackTableVisionJob30.jobStatus.completed;
   IF #_w1 THEN "Unit1.Em6.ControlNodes".stackTable.jobInterface.visionJob30.workingDone := TRUE; END_IF;
   #_w2 := #instStackTableDownJob31.jobStatus.completed AND NOT #statPulse.workingDone[31];   // rising edge of #instStackTableDownJob31.jobStatus.completed
   #statPulse.workingDone[31] := #instStackTableDownJob31.jobStatus.completed;
   #statTonTime[3].TON(IN := (NOT #statUnitStatus.specialFunctions.dryRun AND "Unit1.Em6.ControlNodes".cm.softCam.stackTableAxisZ.currentJRThickness.inPos) OR (#statUnitStatus.specialFunctions.dryRun AND #statUnitStatus.state.idle),
                       PT := T#1000ms);
   #_w3 := #statTonTime[3].Q AND NOT #statPulse.workingDone[32];   // rising edge
   #statPulse.workingDone[32] := #statTonTime[3].Q;
   IF #_w2 OR #_w3 THEN
       "Unit1.Em6.ControlNodes".stackTable.jobInterface.visionJob30.workingDone := FALSE;
   END_IF;
   "Unit1.Em6.ControlNodes".stackTable.jobInterface.tableDownJob31.workingDone := #instStackTableDownJob31.jobStatus.completed;
END_REGION

REGION Network 39: Stack Table Job Interface Working Done [04]
   RUNG wire#powerrail
      Contact( #instStackTableUnloadJob4.jobStatus.completed )
      Coil( "Unit1.Em6.ControlNodes".stackTable.jobInterface.unloadJob4.workingDone )
   END_RUNG
   // the same network as SCL:
   "Unit1.Em6.ControlNodes".stackTable.jobInterface.unloadJob4.workingDone := #instStackTableUnloadJob4.jobStatus.completed;
END_REGION

REGION Network 40: Stack Table Previous Operation Check
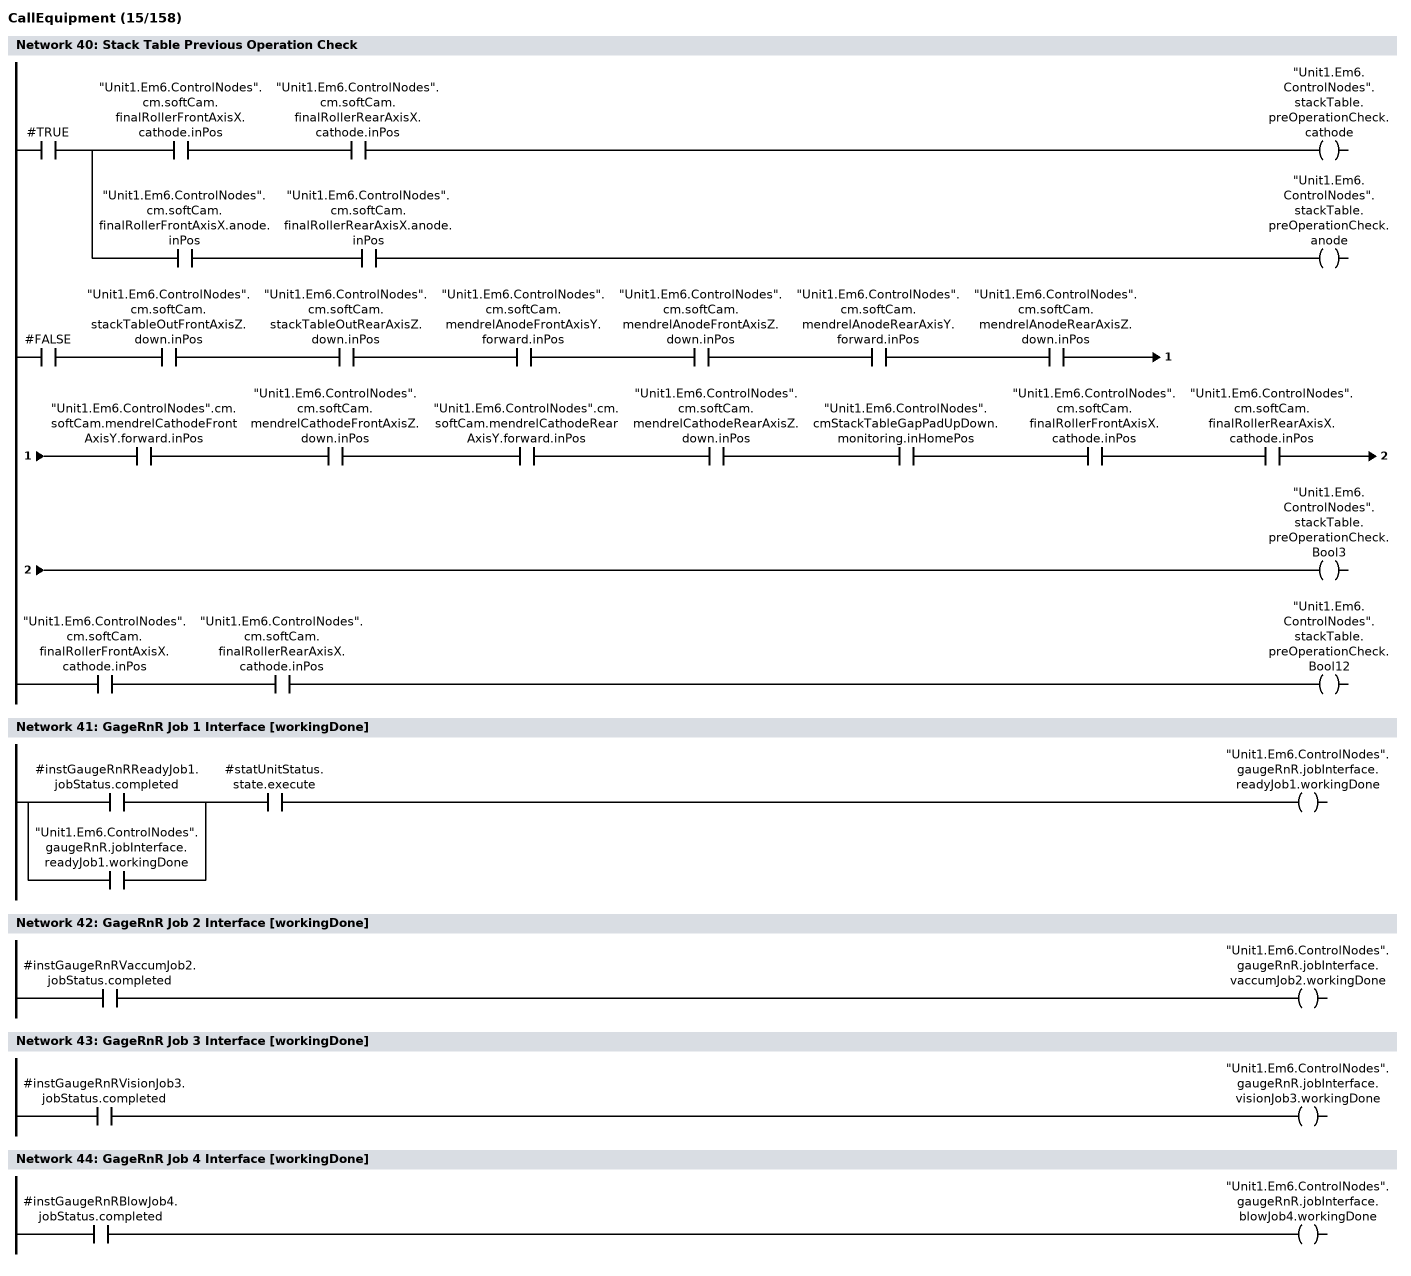
   RUNG wire#powerrail
      Contact( #TRUE )
      wire#w1
      Contact( "Unit1.Em6.ControlNodes".cm.softCam.finalRollerFrontAxisX.cathode.inPos )
      Contact( "Unit1.Em6.ControlNodes".cm.softCam.finalRollerRearAxisX.cathode.inPos )
      Coil( "Unit1.Em6.ControlNodes".stackTable.preOperationCheck.cathode )
   END_RUNG
   RUNG wire#w1
      Contact( "Unit1.Em6.ControlNodes".cm.softCam.finalRollerFrontAxisX.anode.inPos )
      Contact( "Unit1.Em6.ControlNodes".cm.softCam.finalRollerRearAxisX.anode.inPos )
      Coil( "Unit1.Em6.ControlNodes".stackTable.preOperationCheck.anode )
   END_RUNG
   RUNG wire#powerrail
      Contact( #FALSE )
      Contact( "Unit1.Em6.ControlNodes".cm.softCam.stackTableOutFrontAxisZ.down.inPos )
      Contact( "Unit1.Em6.ControlNodes".cm.softCam.stackTableOutRearAxisZ.down.inPos )
      Contact( "Unit1.Em6.ControlNodes".cm.softCam.mendrelAnodeFrontAxisY.forward.inPos )
      Contact( "Unit1.Em6.ControlNodes".cm.softCam.mendrelAnodeFrontAxisZ.down.inPos )
      Contact( "Unit1.Em6.ControlNodes".cm.softCam.mendrelAnodeRearAxisY.forward.inPos )
      Contact( "Unit1.Em6.ControlNodes".cm.softCam.mendrelAnodeRearAxisZ.down.inPos )
      Contact( "Unit1.Em6.ControlNodes".cm.softCam.mendrelCathodeFrontAxisY.forward.inPos )
      Contact( "Unit1.Em6.ControlNodes".cm.softCam.mendrelCathodeFrontAxisZ.down.inPos )
      Contact( "Unit1.Em6.ControlNodes".cm.softCam.mendrelCathodeRearAxisY.forward.inPos )
      Contact( "Unit1.Em6.ControlNodes".cm.softCam.mendrelCathodeRearAxisZ.down.inPos )
      Contact( "Unit1.Em6.ControlNodes".cmStackTableGapPadUpDown.monitoring.inHomePos )
      Contact( "Unit1.Em6.ControlNodes".cm.softCam.finalRollerFrontAxisX.cathode.inPos )
      Contact( "Unit1.Em6.ControlNodes".cm.softCam.finalRollerRearAxisX.cathode.inPos )
      Coil( "Unit1.Em6.ControlNodes".stackTable.preOperationCheck.Bool3 )
   END_RUNG
   RUNG wire#powerrail
      Contact( "Unit1.Em6.ControlNodes".cm.softCam.finalRollerFrontAxisX.cathode.inPos )
      Contact( "Unit1.Em6.ControlNodes".cm.softCam.finalRollerRearAxisX.cathode.inPos )
      Coil( "Unit1.Em6.ControlNodes".stackTable.preOperationCheck.Bool12 )
   END_RUNG
   // the same network as SCL:
   "Unit1.Em6.ControlNodes".stackTable.preOperationCheck.cathode := #TRUE AND "Unit1.Em6.ControlNodes".cm.softCam.finalRollerFrontAxisX.cathode.inPos AND "Unit1.Em6.ControlNodes".cm.softCam.finalRollerRearAxisX.cathode.inPos;
   "Unit1.Em6.ControlNodes".stackTable.preOperationCheck.anode := #TRUE AND "Unit1.Em6.ControlNodes".cm.softCam.finalRollerFrontAxisX.anode.inPos AND "Unit1.Em6.ControlNodes".cm.softCam.finalRollerRearAxisX.anode.inPos;
   "Unit1.Em6.ControlNodes".stackTable.preOperationCheck.Bool3 := #FALSE AND "Unit1.Em6.ControlNodes".cm.softCam.stackTableOutFrontAxisZ.down.inPos AND "Unit1.Em6.ControlNodes".cm.softCam.stackTableOutRearAxisZ.down.inPos AND "Unit1.Em6.ControlNodes".cm.softCam.mendrelAnodeFrontAxisY.forward.inPos AND "Unit1.Em6.ControlNodes".cm.softCam.mendrelAnodeFrontAxisZ.down.inPos AND "Unit1.Em6.ControlNodes".cm.softCam.mendrelAnodeRearAxisY.forward.inPos AND "Unit1.Em6.ControlNodes".cm.softCam.mendrelAnodeRearAxisZ.down.inPos AND "Unit1.Em6.ControlNodes".cm.softCam.mendrelCathodeFrontAxisY.forward.inPos AND "Unit1.Em6.ControlNodes".cm.softCam.mendrelCathodeFrontAxisZ.down.inPos AND "Unit1.Em6.ControlNodes".cm.softCam.mendrelCathodeRearAxisY.forward.inPos AND "Unit1.Em6.ControlNodes".cm.softCam.mendrelCathodeRearAxisZ.down.inPos AND "Unit1.Em6.ControlNodes".cmStackTableGapPadUpDown.monitoring.inHomePos AND "Unit1.Em6.ControlNodes".cm.softCam.finalRollerFrontAxisX.cathode.inPos AND "Unit1.Em6.ControlNodes".cm.softCam.finalRollerRearAxisX.cathode.inPos;
   "Unit1.Em6.ControlNodes".stackTable.preOperationCheck.Bool12 := "Unit1.Em6.ControlNodes".cm.softCam.finalRollerFrontAxisX.cathode.inPos AND "Unit1.Em6.ControlNodes".cm.softCam.finalRollerRearAxisX.cathode.inPos;
END_REGION

REGION Network 41: GageRnR Job 1 Interface [workingDone]
   RUNG wire#powerrail
      Contact( #instGaugeRnRReadyJob1.jobStatus.completed )
      wire#w1
      Contact( #statUnitStatus.state.execute )
      Coil( "Unit1.Em6.ControlNodes".gaugeRnR.jobInterface.readyJob1.workingDone )
   END_RUNG
   RUNG wire#powerrail
      Contact( "Unit1.Em6.ControlNodes".gaugeRnR.jobInterface.readyJob1.workingDone )
   END_RUNG wire#w1
   // the same network as SCL:
   "Unit1.Em6.ControlNodes".gaugeRnR.jobInterface.readyJob1.workingDone := (#instGaugeRnRReadyJob1.jobStatus.completed OR "Unit1.Em6.ControlNodes".gaugeRnR.jobInterface.readyJob1.workingDone) AND #statUnitStatus.state.execute;
END_REGION

REGION Network 42: GageRnR Job 2 Interface [workingDone]
   RUNG wire#powerrail
      Contact( #instGaugeRnRVaccumJob2.jobStatus.completed )
      Coil( "Unit1.Em6.ControlNodes".gaugeRnR.jobInterface.vaccumJob2.workingDone )
   END_RUNG
   // the same network as SCL:
   "Unit1.Em6.ControlNodes".gaugeRnR.jobInterface.vaccumJob2.workingDone := #instGaugeRnRVaccumJob2.jobStatus.completed;
END_REGION

REGION Network 43: GageRnR Job 3 Interface [workingDone]
   RUNG wire#powerrail
      Contact( #instGaugeRnRVisionJob3.jobStatus.completed )
      Coil( "Unit1.Em6.ControlNodes".gaugeRnR.jobInterface.visionJob3.workingDone )
   END_RUNG
   // the same network as SCL:
   "Unit1.Em6.ControlNodes".gaugeRnR.jobInterface.visionJob3.workingDone := #instGaugeRnRVisionJob3.jobStatus.completed;
END_REGION

REGION Network 44: GageRnR Job 4 Interface [workingDone]
   RUNG wire#powerrail
      Contact( #instGaugeRnRBlowJob4.jobStatus.completed )
      Coil( "Unit1.Em6.ControlNodes".gaugeRnR.jobInterface.blowJob4.workingDone )
   END_RUNG
   // the same network as SCL:
   "Unit1.Em6.ControlNodes".gaugeRnR.jobInterface.blowJob4.workingDone := #instGaugeRnRBlowJob4.jobStatus.completed;
END_REGION

REGION Network 46: EM Status Enabled
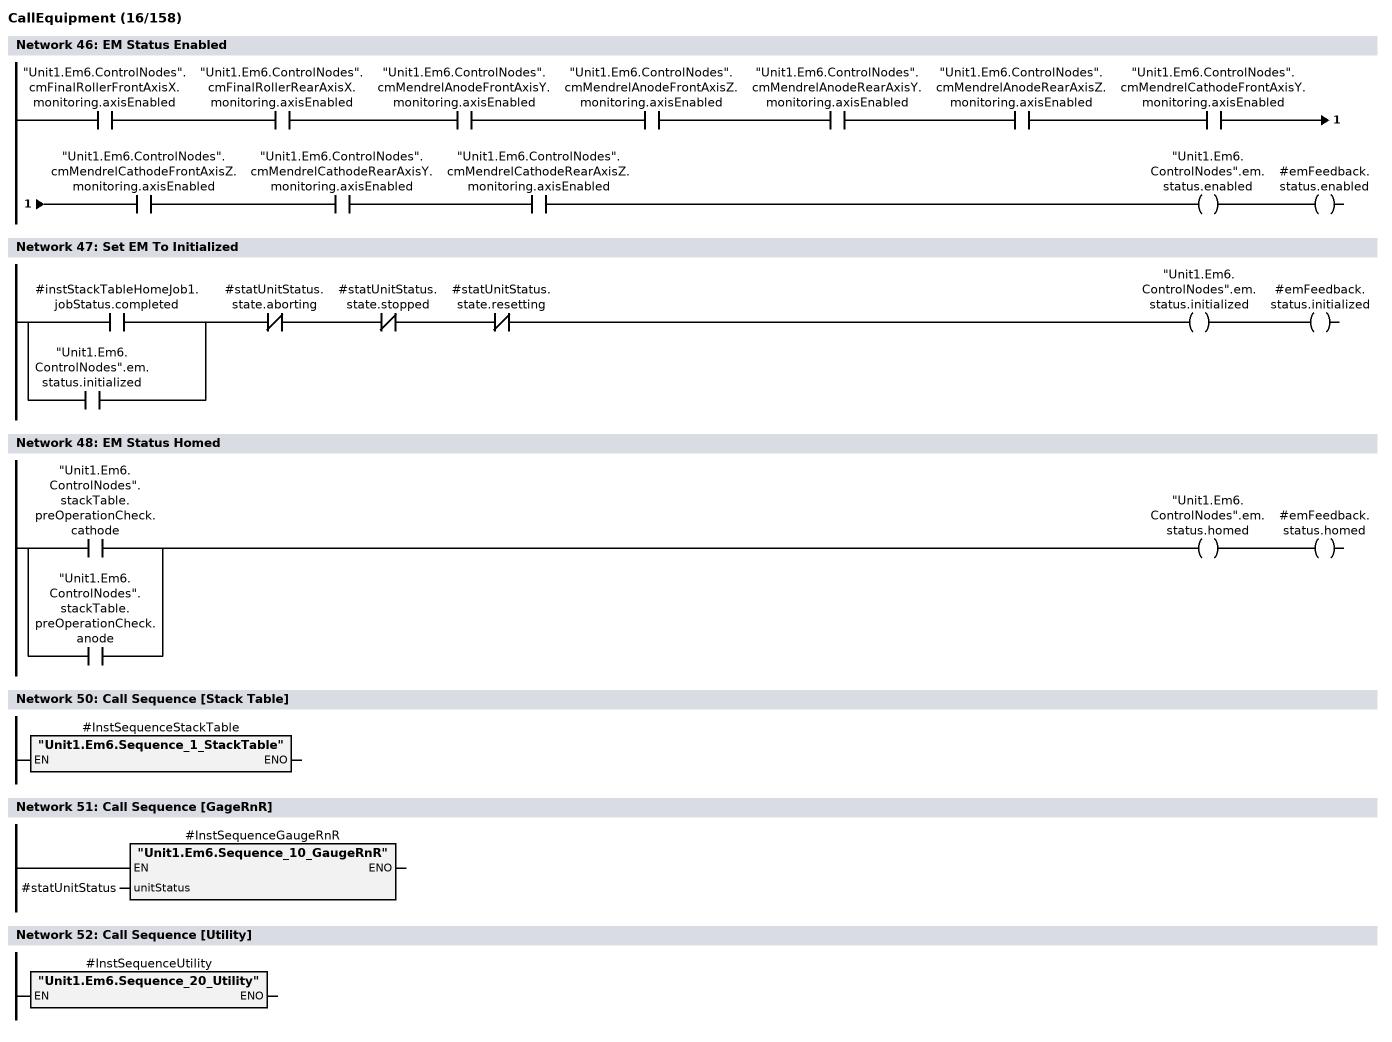
   RUNG wire#powerrail
      Contact( "Unit1.Em6.ControlNodes".cmFinalRollerFrontAxisX.monitoring.axisEnabled )
      Contact( "Unit1.Em6.ControlNodes".cmFinalRollerRearAxisX.monitoring.axisEnabled )
      Contact( "Unit1.Em6.ControlNodes".cmMendrelAnodeFrontAxisY.monitoring.axisEnabled )
      Contact( "Unit1.Em6.ControlNodes".cmMendrelAnodeFrontAxisZ.monitoring.axisEnabled )
      Contact( "Unit1.Em6.ControlNodes".cmMendrelAnodeRearAxisY.monitoring.axisEnabled )
      Contact( "Unit1.Em6.ControlNodes".cmMendrelAnodeRearAxisZ.monitoring.axisEnabled )
      Contact( "Unit1.Em6.ControlNodes".cmMendrelCathodeFrontAxisY.monitoring.axisEnabled )
      Contact( "Unit1.Em6.ControlNodes".cmMendrelCathodeFrontAxisZ.monitoring.axisEnabled )
      Contact( "Unit1.Em6.ControlNodes".cmMendrelCathodeRearAxisY.monitoring.axisEnabled )
      Contact( "Unit1.Em6.ControlNodes".cmMendrelCathodeRearAxisZ.monitoring.axisEnabled )
      Coil( "Unit1.Em6.ControlNodes".em.status.enabled )
      Coil( #emFeedback.status.enabled )
   END_RUNG
   // the same network as SCL:
   "Unit1.Em6.ControlNodes".em.status.enabled := "Unit1.Em6.ControlNodes".cmFinalRollerFrontAxisX.monitoring.axisEnabled AND "Unit1.Em6.ControlNodes".cmFinalRollerRearAxisX.monitoring.axisEnabled AND "Unit1.Em6.ControlNodes".cmMendrelAnodeFrontAxisY.monitoring.axisEnabled AND "Unit1.Em6.ControlNodes".cmMendrelAnodeFrontAxisZ.monitoring.axisEnabled AND "Unit1.Em6.ControlNodes".cmMendrelAnodeRearAxisY.monitoring.axisEnabled AND "Unit1.Em6.ControlNodes".cmMendrelAnodeRearAxisZ.monitoring.axisEnabled AND "Unit1.Em6.ControlNodes".cmMendrelCathodeFrontAxisY.monitoring.axisEnabled AND "Unit1.Em6.ControlNodes".cmMendrelCathodeFrontAxisZ.monitoring.axisEnabled AND "Unit1.Em6.ControlNodes".cmMendrelCathodeRearAxisY.monitoring.axisEnabled AND "Unit1.Em6.ControlNodes".cmMendrelCathodeRearAxisZ.monitoring.axisEnabled;
   #emFeedback.status.enabled := "Unit1.Em6.ControlNodes".em.status.enabled;
END_REGION

REGION Network 47: Set EM To Initialized
   RUNG wire#powerrail
      Contact( #instStackTableHomeJob1.jobStatus.completed )
      wire#w1
      I_Contact( #statUnitStatus.state.aborting )
      I_Contact( #statUnitStatus.state.stopped )
      I_Contact( #statUnitStatus.state.resetting )
      Coil( "Unit1.Em6.ControlNodes".em.status.initialized )
      Coil( #emFeedback.status.initialized )
   END_RUNG
   RUNG wire#powerrail
      Contact( "Unit1.Em6.ControlNodes".em.status.initialized )
   END_RUNG wire#w1
   // the same network as SCL:
   "Unit1.Em6.ControlNodes".em.status.initialized := (#instStackTableHomeJob1.jobStatus.completed OR "Unit1.Em6.ControlNodes".em.status.initialized) AND NOT #statUnitStatus.state.aborting AND NOT #statUnitStatus.state.stopped AND NOT #statUnitStatus.state.resetting;
   #emFeedback.status.initialized := "Unit1.Em6.ControlNodes".em.status.initialized;
END_REGION

REGION Network 48: EM Status Homed
   RUNG wire#powerrail
      Contact( "Unit1.Em6.ControlNodes".stackTable.preOperationCheck.cathode )
      wire#w1
      Coil( "Unit1.Em6.ControlNodes".em.status.homed )
      Coil( #emFeedback.status.homed )
   END_RUNG
   RUNG wire#powerrail
      Contact( "Unit1.Em6.ControlNodes".stackTable.preOperationCheck.anode )
   END_RUNG wire#w1
   // the same network as SCL:
   "Unit1.Em6.ControlNodes".em.status.homed := "Unit1.Em6.ControlNodes".stackTable.preOperationCheck.cathode OR "Unit1.Em6.ControlNodes".stackTable.preOperationCheck.anode;
   #emFeedback.status.homed := "Unit1.Em6.ControlNodes".em.status.homed;
END_REGION

REGION Network 50: Call Sequence [Stack Table]
   RUNG wire#powerrail
      #InstSequenceStackTable()
   END_RUNG
   // the same network as SCL:
   #InstSequenceStackTable();   // "Unit1.Em6.Sequence_1_StackTable"
END_REGION

REGION Network 51: Call Sequence [GageRnR]
   RUNG wire#powerrail
      #InstSequenceGaugeRnR(unitStatus := #statUnitStatus)
   END_RUNG
   // the same network as SCL:
   #InstSequenceGaugeRnR(unitStatus := #statUnitStatus);   // "Unit1.Em6.Sequence_10_GaugeRnR"
END_REGION

REGION Network 52: Call Sequence [Utility]
   RUNG wire#powerrail
      #InstSequenceUtility()
   END_RUNG
   // the same network as SCL:
   #InstSequenceUtility();   // "Unit1.Em6.Sequence_20_Utility"
END_REGION

REGION Network 53: ********** Control Modules (Axis) **********
   // Call control modules that are actuators after the em logic (jobs and sequence), so that the latest commands are applied to the actuators.
END_REGION

